ACTION Ca_StandbySub4:
IF Mach_Control.U.DT_iMode=1 THEN//在自动状态下	
//Ca_Step3-----负极叠片搬运取纠偏位极片
CASE Ca_Step3 OF
	10:
		IF arrAxisCtrl[AxiseNo.AxisName.CaDTCarryingUpDown].Status.Enabled AND arrAxisCtrl[AxiseNo.AxisName.CaDTCarryingLine].Status.Enabled  THEN
			arrCyCtrl[arrCyNo.CylinderName.CaScrapbinCy].Cmd.bON:=TRUE;//负极纠偏NG料盒气缸伸出
			IF arrCyCtrl[arrCyNo.CylinderName.CaScrapbinCy].Status.ONState THEN
				arrCyCtrl[arrCyNo.CylinderName.CaScrapbinUDCy].Cmd.bOFF:=TRUE;//负极纠偏NG料盒气缸升降气缸下降
				IF  arrCyCtrl[arrCyNo.CylinderName.CaScrapbinUDCy].Status.OFFState THEN
					Ca_Step3:=11;
				END_IF
			END_IF	
		END_IF
	11://判断负极搬运平移2是否在初始位，负极搬运升降2上升至初始高度、负极叠片升降上升至初始高度
		IF arrAxisCtrl[AxiseNo.AxisName.CaDTCarryingLine].Cmd.arrbRealPoint[1] THEN
			IF Mach_Control.DT_b.SinStepMode THEN//单步调试模式
				DP_SinStepe:=TRUE;
			ELSE
				DP_SinStepe:=FALSE;	
			END_IF			
			Ca_Step3:=30;
		ELSE
			IF arrAxisCtrl[AxiseNo.AxisName.CaDTCarryingUpDown].Status.Homed AND arrAxisCtrl[AxiseNo.AxisName.CaDTCarryingUpDown].Status.NoMoving AND
				NOT arrAxisCtrl[AxiseNo.AxisName.CaDTCarryingUpDown].Status.Error THEN
				IF arrAxisCtrl[AxiseNo.AxisName.CaDTCarryingUpDown].Cmd.arrbRealPoint[4] THEN
					arrAxisCtrl[AxiseNo.AxisName.CaDTCarryingUpDown].Cmd.iGoSetPos:=0;
					IF Mach_Control.DT_b.SinStepMode THEN//单步调试模式
						DP_SinStepe:=TRUE;
					ELSE
						DP_SinStepe:=FALSE;	
					END_IF								
					Ca_Step3:=20;
				ELSE
					arrAxisCtrl[AxiseNo.AxisName.CaDTCarryingUpDown].Cmd.iGoSetPos:=4;//负极叠片升降移动至等待高度
				END_IF
			END_IF
		END_IF
	20://负极叠片搬运平移至初始位，负极搬运在安全位
		//IF arrAxisCtrl[AxiseNo.AxisName.CaDTCarryingLine].Status.fActPos < (arrAxisPar[AxiseNo.AxisName.CaDTCarryingLine].arrTargetPoint[2]-180) THEN
			//arrCyCtrl[arrCyNo.ElectValveName.CadeviationIonizedWind].Cmd.bON:=TRUE;//负极纠偏平台除尘
			//arrCyCtrl[arrCyNo.ElectValveName.CadeviationIonizedWind].Cmd.bOFF:=FALSE;//负极纠偏平台除尘
		//END_IF	
		IF NOT DP_SinStepe THEN
			//arrCyCtrl[arrCyNo.CylinderName.CaScrapbinCy].Cmd.bOFF:=TRUE;//负极纠偏NG料盒气缸收回   Mach_Control.Ca_b.CarryingSafepos[0] 
			IF TailCurlSEPTA_SafePos AND arrAxisCtrl[AxiseNo.AxisName.CaCarryingUpDown2].Cmd.arrbRealPoint[4] AND arrAxisCtrl[AxiseNo.AxisName.CaDTCarryingUpDown].Cmd.arrbRealPoint[4] AND arrAxisCtrl[AxiseNo.AxisName.CaDTCarryingLine].Status.Homed AND
				arrAxisCtrl[AxiseNo.AxisName.CaDTCarryingLine].Status.NoMoving AND NOT arrAxisCtrl[AxiseNo.AxisName.CaDTCarryingLine].Status.Error (*AND NOT arrAxisCtrl[AxiseNo.AxisName.CaCarryingLine2].Status.Error AND
				arrAxisCtrl[AxiseNo.AxisName.CaCarryingLine2].Status.fActPos < arrAxisPar[AxiseNo.AxisName.CaCarryingLine2].arrTargetPoint[2]*)    THEN
				IF arrAxisCtrl[AxiseNo.AxisName.CaDTCarryingLine].Cmd.arrbRealPoint[1] THEN
					Ca_DTCarryingTorMark:=FALSE;//负极叠台搬运平移力矩判断标志位
					arrAxisCtrl[AxiseNo.AxisName.CaDTCarryingLine].Cmd.iGoSetPos:=0;
					IF Mach_Control.DT_b.SinStepMode THEN//单步调试模式
						DP_SinStepe:=TRUE;
					ELSE
						DP_SinStepe:=FALSE;	
					END_IF					
					Ca_Step3:=30;
				ELSE
					arrAxisCtrl[AxiseNo.AxisName.CaDTCarryingLine].Cmd.iGoSetPos:=1;//负极叠片平移至初始位
					Ca_DTCarryingTorMark:=TRUE;//负极叠台搬运平移力矩判断标志位
				END_IF
			END_IF
		END_IF
	30://判断纠偏平台是否允许取极片
		IF NOT DP_SinStepe THEN
			IF 	Mach_Control.Ca_b.Ca_deviationDPOK OR Mach_Control.U.EmptyRunMode  THEN
				IF Mach_Control.DT_b.SinStepMode THEN//单步调试模式
					DP_SinStepe:=TRUE;
				ELSE
					DP_SinStepe:=FALSE;	
				END_IF			
				IF Mach_Control.DT_b.DT_CCD_TwoModel THEN
					CCD.CaRec.Finish.RectifyX1:=0;
					CCD.CaRec.Finish.RectifyX2:=0;
					CCD.CaRec.Finish.RectifyY:=0;		
					CCD.CaRec.Finish.RectifyResult:=0;//拍照结果清零									
					Mach_Control.Ca_b.Ca_CCDStart :=TRUE;//启动CCD拍照
					CCD.CaRec.Start.iPhotoDo:=2;//启动CCD第二次拍照
				END_IF		
				Ca_TON[7].IN:=FALSE;
				Ca_Step3:=40;
			END_IF
		END_IF
	
END_CASE
END_IF



CASE Ca_Step3 OF

	40://AND  arrCyCtrl[arrCyNo.CylinderName.CaScrapbinCy].Io.DIOFFSwitch  arrCyCtrl[arrCyNo.CylinderName.CaScrapbinCy].Io.DIOFFSwitch AND						
		IF NOT DP_SinStepe THEN
			arrCyCtrl[arrCyNo.ElectValveName.CaDTCarryingVacuum].Cmd.bON:=FALSE;//负极叠片搬运升降真空开
			arrCyCtrl[arrCyNo.ElectValveName.CaDTCarryingVacuum].Cmd.bOFF:=TRUE;//负极叠片搬运升降真空开
	
			//arrCyCtrl[arrCyNo.CylinderName.CaScrapbinCy].Cmd.bOFF:=TRUE;//负极纠偏NG料盒气缸收回
			IF  arrAxisCtrl[AxiseNo.AxisName.CaDTCarryingUpDown].Status.Homed AND 
				arrAxisCtrl[AxiseNo.AxisName.CaDTCarryingUpDown].Status.NoMoving AND NOT arrAxisCtrl[AxiseNo.AxisName.CaDTCarryingUpDown].Status.Error THEN
				IF arrAxisCtrl[AxiseNo.AxisName.CaDTCarryingUpDown].Cmd.arrbRealPoint[2] AND arrCyCtrl[arrCyNo.CylinderName.CaScrapbinCy].Status.ONState THEN
					arrCyCtrl[arrCyNo.ElectValveName.CadeviationVacuum].Cmd.bOFF:=TRUE;//负极纠偏平台真空关闭
					arrCyCtrl[arrCyNo.ElectValveName.CadeviationVacuum].Cmd.bON:=FALSE;//负极纠偏平台真空关闭
					arrCyCtrl[arrCyNo.ElectValveName.CadeviationVacuumBark].Cmd.bON:=TRUE;//负极纠偏平台破真空打开	
					arrCyCtrl[arrCyNo.ElectValveName.CadeviationVacuumBark].Cmd.bOFF:=FALSE;//负极纠偏平台破真空打开		
					//IF Mach_Control.Ca_b.Ca_deviationFalg THEN
						Mach_Control.Ca_b.Ca_DPCarryingFalg:=TRUE;//置位叠片真空吸盘有料标记	
						Mach_Control.Ca_b.Ca_deviationFalg:=FALSE;//复位纠偏平台有料标记			
					//END_IF
					Par.stDT_date.Ca_MQ_Slice[9]:=Par.stDT_date.Ca_MQ_Slice[8];											
					arrAxisCtrl[AxiseNo.AxisName.CaDTCarryingUpDown].Cmd.iGoSetPos:=0;									
					IF NOT Ca_TON[7].Q THEN
						Ca_TON[7].IN:=TRUE;
					ELSE
						IF Mach_Control.DT_b.SinStepMode THEN//单步调试模式
							DP_SinStepe:=TRUE;
						ELSE
							DP_SinStepe:=FALSE;	
						END_IF			
						Ca_TON[7].IN:=FALSE;
						Ca_Step3:=50;												
					END_IF												
				ELSE
					arrAxisCtrl[AxiseNo.AxisName.CaDTCarryingUpDown].Cmd.iGoSetPos:=2;//负极叠片升降下降至取纠偏极片高度
				END_IF
			END_IF	
		END_IF
	50://负极叠片搬运升降上升至凸轮耦合初始位
		IF arrAxisCtrl[AxiseNo.AxisName.CaDTCarryingUpDown].Status.Homed AND arrAxisCtrl[AxiseNo.AxisName.CaDTCarryingUpDown].Status.NoMoving AND 
			NOT arrAxisCtrl[AxiseNo.AxisName.CaDTCarryingUpDown].Status.Error THEN
				IF arrAxisCtrl[AxiseNo.AxisName.CaDTCarryingUpDown].Cmd.arrbRealPoint[4] THEN
					arrAxisCtrl[AxiseNo.AxisName.CaDTCarryingUpDown].Cmd.iGoSetPos:=0;
					Ca_Step3:=6666;
				ELSE
					arrAxisCtrl[AxiseNo.AxisName.CaDTCarryingUpDown].Cmd.iGoSetPos:=4;//负极叠片升降移动至初始高度
				END_IF
		END_IF		
END_CASE
END_ACTION

ACTION Code:
(*
 TJ_Scan_M(CLK:=Mach_Control.TJ_b.Scan_CT , Q=> );
 CASE scan_Step OF
	0:
		IF TJ_Scan_M.Q THEN
			scan_Step:=5;
		END_IF
	5:
		 Mach_Control.TJ_b.Scan_Men[4]:=Mach_Control.TJ_b.Scan_Men[3];
		 scan_Step:=10;
	 
	10:
		Mach_Control.TJ_b.Scan_Men[3]:=Mach_Control.TJ_b.Scan_Men[2];
	 	scan_Step:=20;
	 
	 20:
	 	Mach_Control.TJ_b.Scan_Men[2]:=Mach_Control.TJ_b.Scan_Men[1];
	 	scan_Step:=30;
	 
	 30:
	 		Mach_Control.TJ_b.Scan_Men[1].Scan_gross:=Mach_Control.TJ_b.Scan_gross;
	 		Mach_Control.TJ_b.Scan_Men[1].TJ_Code:=Mach_Control.TJ_b.strCode;
	 		scan_Step:=0;
	 
	 
 END_CASE
 *)
END_ACTION

ACTION Dietai_Cam:
DT_Cam_ton[1](PT:=T#100MS);
DT_Cam_ton[2](PT:=T#100MS);
DT_Cam_ton[3](PT:=T#100MS);
DT_Cam_ton[4](PT:=T#100MS);
DT_Cam_ton[5](PT:=T#100MS);
DT_Cam_ton[5](PT:=T#100MS);//
(***********************************压刀凸轮表创建************************************************)
(*
    fbCrectCamLeftYDLine                   :FB_CrectCamYaDaoLine ;
     fbCrectCamLeftYDUpDown             :FB_CrectCamYaDaoUpDown ;
     fbCrectCamRightYDLine                 :FB_CrectCamYaDaoLine ;
     fbCrectCamRightYDUpDown           :FB_CrectCamYaDaoUpDown ;
*)
//左压刀升降凸轮创建 
//fbCrectCamLeftYDUpDown.fMoveLength:=-ABS(arrAxisPar[AxiseNo.AxisName.LeftYDUpDown].arrTargetPoint[1]-arrAxisPar[AxiseNo.AxisName.LeftYDUpDown].arrTargetPoint[2]);
//fbCrectCamLeftYDUpDown.fSaveLength1:=-ABS(arrAxisPar[AxiseNo.AxisName.LeftYDUpDown].arrTargetPoint[1]-arrAxisPar[AxiseNo.AxisName.LeftYDUpDown].arrTargetPoint[3]);
fbCrectCamLeftYDUpDown.fMoveLength:=-ABS(arrAxisPar[AxiseNo.AxisName.LeftYDUpDown].arrTargetPoint[11]+arrAxisPar[AxiseNo.AxisName.LeftYDUpDown].arrTargetPoint[13]);
fbCrectCamLeftYDUpDown.fSaveLength1:=-ABS(arrAxisPar[AxiseNo.AxisName.LeftYDUpDown].arrTargetPoint[12]+arrAxisPar[AxiseNo.AxisName.LeftYDUpDown].arrTargetPoint[13]);
fbCrectCamLeftYDUpDown.fSaveLength2:=-3;

fbCrectCamLeftYDUpDown(
	bCreatTable:=                       fbCrectCamLeftYDUpDown.bCreatTable , 
	Reset:=                                 stSysState.bReset  ,  
	iTable:=                                TableNo.M_LeftYDUpDown  , 
	fMoveLength:=  , //压刀升降最大高度
	fSaveLength1:= , //压刀抽刀高度
	fSaveLength2:= , //压刀下压高度
	fMasterKeyPos1:=240 , //220 240
	fMasterKeyPos2:=258 , //234 250
	fMasterKeyPos3:=275 , //252 255
	fMasterKeyPos4:=307 , //300
	//fMasterKeyPos5:=313 , //330
	fMasterKeyPos6:=342 , //342
    axisMaster:=                          arrAxis[AxiseNo.VirAxisName.VirMain] ,   
	axisSlave:=                             arrAxis[AxiseNo.AxisName.LeftYDUpDown] ,  
	
	bCreatTableDone=> , 
	bCreatTableError=> , 
	bError=> );
fbCrectCamLeftYDUpDown.bCreatTableDone;
fbCrectCamLeftYDUpDown.bCreatTableError;
fbCrectCamLeftYDUpDown.bError;

//左压刀开合凸轮创建
//fbCrectCamLeftYDLine.fMoveLength:=-ABS(arrAxisPar[AxiseNo.AxisName.LeftYDLine].arrTargetPoint[1]-arrAxisPar[AxiseNo.AxisName.LeftYDLine].arrTargetPoint[2]);
fbCrectCamLeftYDLine.fMoveLength:=-ABS(arrAxisPar[AxiseNo.AxisName.LeftYDLine].arrTargetPoint[11]);
fbCrectCamLeftYDLine.fMoveLength2:=-ABS(arrAxisPar[AxiseNo.AxisName.LeftYDLine].arrTargetPoint[12]);	
fbCrectCamLeftYDLine(
	bCreatTable:=                         fbCrectCamLeftYDLine.bCreatTable , 
	Reset:=                                   stSysState.bReset  ,  
	iTable:=                                   TableNo.M_LeftYDLine  , 
	fMoveLength:= , 
	fMasterKeyPos1:=260 , //234  250
	fMasterKeyPos4:=40 , //234  250
	fMasterKeyPos2:=293 , //290
	fMasterKeyPos3:=328 , //324
	axisMaster:=                       arrAxis[AxiseNo.VirAxisName.VirMain] ,   
    axisSlave:=                          arrAxis[AxiseNo.AxisName.LeftYDLine] ,  
	bCreatTableDone=>  , 
	bCreatTableError=> , 
	bError=> );
fbCrectCamLeftYDLine.bCreatTableDone;
fbCrectCamLeftYDLine.bCreatTableError;
fbCrectCamLeftYDLine.bError;

//右压刀开合
//fbCrectCamRightYDLine.fMoveLength:=-ABS(arrAxisPar[AxiseNo.AxisName.RightYDLine].arrTargetPoint[1]-arrAxisPar[AxiseNo.AxisName.RightYDLine].arrTargetPoint[2]);
fbCrectCamRightYDLine.fMoveLength:=-ABS(arrAxisPar[AxiseNo.AxisName.RightYDLine].arrTargetPoint[11]);
fbCrectCamRightYDLine.fMoveLength2:=-ABS(arrAxisPar[AxiseNo.AxisName.RightYDLine].arrTargetPoint[12]);
fbCrectCamRightYDLine(
	bCreatTable:=                         fbCrectCamRightYDLine.bCreatTable , 
	Reset:=                                   stSysState.bReset  ,  
	iTable:=                                   TableNo.M_RightYDLine  , 
	fMoveLength:= , 

	fMasterKeyPos1:=260 , //234  250
	fMasterKeyPos4:=40 , //234  250
	fMasterKeyPos2:=293 ,//290
	fMasterKeyPos3:=328 , //324

	axisMaster:=                       arrAxis[AxiseNo.VirAxisName.VirMain] ,   
    axisSlave:=                          arrAxis[AxiseNo.AxisName.RightYDLine] ,  
	bCreatTableDone=>  , 
	bCreatTableError=> , 
	bError=> );
fbCrectCamRightYDLine.bCreatTableDone;
fbCrectCamRightYDLine.bCreatTableError;
fbCrectCamRightYDLine.bError;

//右压刀升降凸轮创建
//fbCrectCamRightYDUpDown.fMoveLength:=-ABS(arrAxisPar[AxiseNo.AxisName.RightYDUpDown].arrTargetPoint[1]-arrAxisPar[AxiseNo.AxisName.RightYDUpDown].arrTargetPoint[2]);
//fbCrectCamRightYDUpDown.fSaveLength1:=-ABS(arrAxisPar[AxiseNo.AxisName.RightYDUpDown].arrTargetPoint[1]-arrAxisPar[AxiseNo.AxisName.RightYDUpDown].arrTargetPoint[3]);
fbCrectCamRightYDUpDown.fMoveLength:=-ABS(arrAxisPar[AxiseNo.AxisName.RightYDUpDown].arrTargetPoint[11]+arrAxisPar[AxiseNo.AxisName.RightYDUpDown].arrTargetPoint[13]);
fbCrectCamRightYDUpDown.fSaveLength1:=-ABS(arrAxisPar[AxiseNo.AxisName.RightYDUpDown].arrTargetPoint[12]+arrAxisPar[AxiseNo.AxisName.RightYDUpDown].arrTargetPoint[13]);	
fbCrectCamRightYDUpDown.fSaveLength2:=-3;
fbCrectCamRightYDUpDown(
	bCreatTable:=                       fbCrectCamRightYDUpDown.bCreatTable , 
	Reset:=                                 stSysState.bReset  ,  
	iTable:=                                TableNo.M_RightYDUpDown  , 
	fMoveLength:= , 
	fSaveLength1:= , 
	fSaveLength2:= ,
	fMasterKeyPos1:=240 , //220 240
	fMasterKeyPos2:=258 , //234 250
	fMasterKeyPos3:=275 , //252 255
	fMasterKeyPos4:=307 , //300
	//fMasterKeyPos5:=313 , //330
	fMasterKeyPos6:=342 , //342
    axisMaster:=                          arrAxis[AxiseNo.VirAxisName.VirMain] ,   
	axisSlave:=                             arrAxis[AxiseNo.AxisName.RightYDUpDown] ,  
	
	bCreatTableDone=> , 
	bCreatTableError=> , 
	bError=> );
fbCrectCamRightYDUpDown.bCreatTableDone;
fbCrectCamRightYDUpDown.bCreatTableError;
fbCrectCamRightYDUpDown.bError;


//左压刀升降凸轮创建 2
fbCrectCamLeftYDUpDown2.fMoveLength:=-ABS(arrAxisPar[AxiseNo.AxisName.LeftYDUpDown].arrTargetPoint[11]+arrAxisPar[AxiseNo.AxisName.LeftYDUpDown].arrTargetPoint[13]);
fbCrectCamLeftYDUpDown2.fSaveLength1:=-ABS(arrAxisPar[AxiseNo.AxisName.LeftYDUpDown].arrTargetPoint[11]+arrAxisPar[AxiseNo.AxisName.LeftYDUpDown].arrTargetPoint[13]);
fbCrectCamLeftYDUpDown2.fSaveLength2:=ABS(arrAxisPar[AxiseNo.AxisName.LeftYDUpDown].arrTargetPoint[12]+arrAxisPar[AxiseNo.AxisName.LeftYDUpDown].arrTargetPoint[13]);
fbCrectCamLeftYDUpDown2(
	bCreatTable:=                       fbCrectCamLeftYDUpDown2.bCreatTable , 
	Reset:=                                 stSysState.bReset  ,  
	iTable:=                                TableNo.M_LeftYDUpDown2  , 
	fMoveLength:=  , //压刀升降最大高度
	fSaveLength1:= , //压刀抽刀高度
	fSaveLength2:= , //
	fMasterKeyPos1:=260 , //240
	fMasterKeyPos2:=300 , //234 250
	fMasterKeyPos3:=301 , //252 255
	fMasterKeyPos4:=302 , //300
//	fMasterKeyPos5:=342 , //300
    fMasterKeyPos6:=342 , //342
    axisMaster:=                          arrAxis[AxiseNo.VirAxisName.VirMain] ,   
	axisSlave:=                             arrAxis[AxiseNo.AxisName.LeftYDUpDown] ,  
	
	bCreatTableDone=> , 
	bCreatTableError=> , 
	bError=> );
fbCrectCamLeftYDUpDown2.bCreatTableDone;
fbCrectCamLeftYDUpDown2.bCreatTableError;
fbCrectCamLeftYDUpDown.bError;

//左压刀开合凸轮创建2

fbCrectCamLeftYDLine2.fMoveLength:=ABS(arrAxisPar[AxiseNo.AxisName.LeftYDLine].arrTargetPoint[1]-arrAxisPar[AxiseNo.AxisName.LeftYDLine].arrTargetPoint[2]);
fbCrectCamLeftYDLine2(
	bCreatTable:=                         fbCrectCamLeftYDLine2.bCreatTable , 
	Reset:=                                   stSysState.bReset  ,  
	iTable:=                                   TableNo.M_LeftYDLine2  , 
	fMoveLength:= , 
	fMasterKeyPos1:=285 , //234  250
	fMasterKeyPos4:=40 , //234  250
	fMasterKeyPos2:=293 , //290
	fMasterKeyPos3:=328 , //324
	axisMaster:=                       arrAxis[AxiseNo.VirAxisName.VirMain] ,   
    axisSlave:=                          arrAxis[AxiseNo.AxisName.LeftYDLine] ,  
	bCreatTableDone=>  , 
	bCreatTableError=> , 
	bError=> );
fbCrectCamLeftYDLine2.bCreatTableDone;
fbCrectCamLeftYDLine2.bCreatTableError;
fbCrectCamLeftYDLine2.bError;


//右压刀开合2

fbCrectCamRightYDLine2.fMoveLength:=ABS(arrAxisPar[AxiseNo.AxisName.RightYDLine].arrTargetPoint[1]-arrAxisPar[AxiseNo.AxisName.RightYDLine].arrTargetPoint[2]);
fbCrectCamRightYDLine2(
	bCreatTable:=                         fbCrectCamRightYDLine2.bCreatTable , 
	Reset:=                                   stSysState.bReset  ,  
	iTable:=                                   TableNo.M_RightYDLine2  , 
	fMoveLength:= , 

	fMasterKeyPos1:=285 , //234  250
	fMasterKeyPos4:=40 , //234  250
	fMasterKeyPos2:=293 ,//290
	fMasterKeyPos3:=328 , //324

	axisMaster:=                       arrAxis[AxiseNo.VirAxisName.VirMain] ,   
    axisSlave:=                          arrAxis[AxiseNo.AxisName.RightYDLine] ,  
	bCreatTableDone=>  , 
	bCreatTableError=> , 
	bError=> );
fbCrectCamRightYDLine2.bCreatTableDone;
fbCrectCamRightYDLine2.bCreatTableError;
fbCrectCamRightYDLine2.bError;

//右压刀升降凸轮创建2
fbCrectCamRightYDUpDown2.fMoveLength:=-ABS(arrAxisPar[AxiseNo.AxisName.RightYDUpDown].arrTargetPoint[11]+arrAxisPar[AxiseNo.AxisName.RightYDUpDown].arrTargetPoint[13]);
fbCrectCamRightYDUpDown2.fSaveLength1:=-ABS(arrAxisPar[AxiseNo.AxisName.RightYDUpDown].arrTargetPoint[11]+arrAxisPar[AxiseNo.AxisName.RightYDUpDown].arrTargetPoint[13]);	
fbCrectCamRightYDUpDown2.fSaveLength2:=ABS(arrAxisPar[AxiseNo.AxisName.RightYDUpDown].arrTargetPoint[12]+arrAxisPar[AxiseNo.AxisName.RightYDUpDown].arrTargetPoint[13]);
fbCrectCamRightYDUpDown2(
	bCreatTable:=                       fbCrectCamRightYDUpDown2.bCreatTable , 
	Reset:=                                 stSysState.bReset  ,  
	iTable:=                                TableNo.M_RightYDUpDown2  , 
	fMoveLength:= , 
	fSaveLength1:= , 
	fSaveLength2:= ,
	fMasterKeyPos1:=260 , //240
	fMasterKeyPos2:=300 , //234 250
	fMasterKeyPos3:=301 , //252 255
	fMasterKeyPos4:=302 , //300
//	fMasterKeyPos5:=342 , //300
    fMasterKeyPos6:=342 , //342
    axisMaster:=                          arrAxis[AxiseNo.VirAxisName.VirMain] ,   
	axisSlave:=                             arrAxis[AxiseNo.AxisName.RightYDUpDown] ,  
	
	bCreatTableDone=> , 
	bCreatTableError=> , 
	bError=> );
fbCrectCamRightYDUpDown2.bCreatTableDone;
fbCrectCamRightYDUpDown2.bCreatTableError;
fbCrectCamRightYDUpDown2.bError;

tYDCreateCamTON(IN:= , PT:=T#0.5S , Q=> , ET=> );
IF Mach_Control.U.DT_iMode=3 OR Mach_Control.U.DT_iMode=0 THEN//在手动状态下
			//从触摸屏创建叠台压刀凸轮
			rYDCreateCam_TRIG(CLK:=Mach_Control.DT_b.CreateCamStart1 , Q=> );		
			IF rYDCreateCam_TRIG.Q THEN
				tYDCreateCamTON.IN:=FALSE;
				YDCrectCamStep0:=10;
				Mach_Control.DT_b.Error[0]:=FALSE;
			END_IF
END_IF			
			//叠台压刀凸轮自动创建
			CASE YDCrectCamStep0 OF
					10:
							IF NOT 	tYDCreateCamTON.Q THEN
									fbCrectCamLeftYDUpDown.bCreatTable:=FALSE;;//左压刀升降凸轮创建
									fbCrectCamLeftYDLine.bCreatTable:=FALSE;//左压刀开合凸轮创建
									fbCrectCamRightYDLine.bCreatTable :=FALSE;//右压刀开合凸轮创建
									 fbCrectCamRightYDUpDown.bCreatTable:=FALSE;//右压刀升降凸轮创建
									 Mach_Control.DT_b.CreateCamDone1:=FALSE;	
									 tYDCreateCamTON.IN:=TRUE;				
							ELSE
										tYDCreateCamTON.IN:=FALSE;
										YDCrectCamStep0:=11;
							END_IF
							
					11:
							IF  NOT DT_Cam_ton[1].Q THEN
								arrAxisCtrl[AxiseNo.AxisName.LeftYDLine].Cmd.bStop:=TRUE;
								arrAxisCtrl[AxiseNo.AxisName.LeftYDUpDown].Cmd.bStop:=TRUE;
								arrAxisCtrl[AxiseNo.AxisName.RightYDLine].Cmd.bStop:=TRUE;
								arrAxisCtrl[AxiseNo.AxisName.RightYDUpDown].Cmd.bStop:=TRUE;
								DT_Cam_ton[1].IN:=TRUE;
							ELSE
								DT_Cam_ton[1].IN:=FALSE;
								YDCrectCamStep0:=12;
								arrAxisCtrl[AxiseNo.AxisName.LeftYDLine].Cmd.bStop:=FALSE;
								arrAxisCtrl[AxiseNo.AxisName.LeftYDUpDown].Cmd.bStop:=FALSE;
								arrAxisCtrl[AxiseNo.AxisName.RightYDLine].Cmd.bStop:=FALSE;
								arrAxisCtrl[AxiseNo.AxisName.RightYDUpDown].Cmd.bStop:=FALSE;
							END_IF
					
					12:
						IF  NOT DT_Cam_ton[2].Q THEN
							arrAxisCtrl[AxiseNo.AxisName.LeftYDLine].Cmd.bReset:=TRUE;	
							arrAxisCtrl[AxiseNo.AxisName.LeftYDUpDown].Cmd.bReset:=TRUE;
							arrAxisCtrl[AxiseNo.AxisName.RightYDLine].Cmd.bReset:=TRUE;
							arrAxisCtrl[AxiseNo.AxisName.RightYDUpDown].Cmd.bReset:=TRUE;		
							DT_Cam_ton[2].IN:=TRUE;
						 ELSE
							 DT_Cam_ton[2].IN:=FALSE;
							 YDCrectCamStep0:=13;
							arrAxisCtrl[AxiseNo.AxisName.LeftYDLine].Cmd.bReset:=FALSE;	
							arrAxisCtrl[AxiseNo.AxisName.LeftYDUpDown].Cmd.bReset:=FALSE;
							arrAxisCtrl[AxiseNo.AxisName.RightYDLine].Cmd.bReset:=FALSE;
							arrAxisCtrl[AxiseNo.AxisName.RightYDUpDown].Cmd.bReset:=FALSE;	
						 END_IF
							
					13:
						arrAxisCtrl[AxiseNo.AxisName.LeftYDLine].Cmd.bEnable:=TRUE;
						arrAxisCtrl[AxiseNo.AxisName.LeftYDUpDown].Cmd.bEnable:=TRUE;
						arrAxisCtrl[AxiseNo.AxisName.RightYDLine].Cmd.bEnable:=TRUE;
						arrAxisCtrl[AxiseNo.AxisName.RightYDUpDown].Cmd.bEnable:=TRUE;
						
						IF arrAxisCtrl[AxiseNo.AxisName.LeftYDLine].Status.Enabled AND arrAxisCtrl[AxiseNo.AxisName.LeftYDUpDown].Status.Enabled AND
							arrAxisCtrl[AxiseNo.AxisName.RightYDLine].Status.Enabled AND arrAxisCtrl[AxiseNo.AxisName.RightYDUpDown].Status.Enabled THEN
							 YDCrectCamStep0:=20;
						END_IF		
				
							
					20://创建凸轮
						fbCrectCamLeftYDUpDown.bCreatTable:=TRUE;;//左压刀升降凸轮创建
						fbCrectCamLeftYDLine.bCreatTable:=TRUE;//左压刀开合凸轮创建
						fbCrectCamRightYDLine.bCreatTable :=TRUE;//右压刀开合凸轮创建
						 fbCrectCamRightYDUpDown.bCreatTable:=TRUE;//右压刀升降凸轮创建
						fbCrectCamLeftYDUpDown2.bCreatTable:=TRUE;;//左压刀升降凸轮创建2
						fbCrectCamLeftYDLine2.bCreatTable:=TRUE;//左压刀开合凸轮创建2
						fbCrectCamRightYDLine2.bCreatTable :=TRUE;//右压刀开合凸轮创建2
						 fbCrectCamRightYDUpDown2.bCreatTable:=TRUE;//右压刀升降凸轮创建	2							 
						 Mach_Control.DT_b.CreateCamDone1:=FALSE;
						 YDCrectCamStep0:=30;
					30://等待凸轮创建完成
						IF fbCrectCamLeftYDUpDown.bCreatTableDone AND fbCrectCamLeftYDLine.bCreatTableDone AND fbCrectCamRightYDLine.bCreatTableDone AND fbCrectCamRightYDUpDown.bCreatTableDone AND
                          fbCrectCamLeftYDUpDown2.bCreatTableDone AND fbCrectCamLeftYDLine2.bCreatTableDone AND fbCrectCamRightYDLine2.bCreatTableDone AND fbCrectCamRightYDUpDown2.bCreatTableDone  THEN
								Mach_Control.DT_b.CreateCamDone1:=TRUE;//叠台压凸轮创建完成
								YDCrectCamStep0:=6666;
						ELSE
								IF fbCrectCamLeftYDUpDown.bCreatTableError OR fbCrectCamLeftYDLine.bCreatTableError OR fbCrectCamRightYDLine.bCreatTableError OR fbCrectCamRightYDUpDown.bCreatTableError  OR
                                   fbCrectCamLeftYDUpDown2.bCreatTableError OR fbCrectCamLeftYDLine2.bCreatTableError OR fbCrectCamRightYDLine2.bCreatTableError OR fbCrectCamRightYDUpDown2.bCreatTableError  THEN
									Mach_Control.DT_b.Error[0]:=TRUE;//叠台压刀凸轮创建失败报警
									YDCrectCamStep0:=9999;
								END_IF
						END_IF
			END_CASE


(***********************************压刀凸轮耦合***********************************************)
(*
      fbCamInLeftYDLine                       :FB_CamIn ;    
      fbCamInLeftYDUpDown                :FB_CamIn ;    
      fbCamInRightYDLine                    :FB_CamIn ;    
      fbCamInRightYDUpDown             :FB_CamIn ;    

*)
//左压刀开合凸轮耦合
fbCamInLeftYDLine.ParCamIn.SlaveScaling;
fbCamInLeftYDLine(
	Reset:=                      stSysState.bReset  , 
	bCamInExecute:=       fbCamInLeftYDLine.bCamInExecute, 
	iTable1:=                   TableNo.M_LeftYDLine  , 
	iTable2:=                   TableNo.M_LeftYDLine2, 
	iTableSel:=                 , 
	ParCamIn:= , 
  	axisMaster:=            arrAxis[AxiseNo.VirAxisName.VirMain] ,  
	axisSlave:=               arrAxis[AxiseNo.AxisName.LeftYDLine] ,  
	bError=> , 
	bReady=> , 
	bInSync=> );

Mach_Control.DT_b.Error[12]:=fbCamInLeftYDLine.bError;
fbCamInLeftYDLine.bReady;
fbCamInLeftYDLine.bInSync;

//左压刀升降凸轮耦合
fbCamInLeftYDUpDown.ParCamIn.SlaveScaling;
fbCamInLeftYDUpDown(
	Reset:=                      stSysState.bReset  , 
	bCamInExecute:=       fbCamInLeftYDUpDown.bCamInExecute, 
	iTable1:=                   TableNo.M_LeftYDUpDown  , 
	iTable2:=                   TableNo.M_LeftYDUpDown2 , 
	iTableSel:=                 , 
	ParCamIn:= , 
  	axisMaster:=            arrAxis[AxiseNo.VirAxisName.VirMain] ,  
	axisSlave:=               arrAxis[AxiseNo.AxisName.LeftYDUpDown] ,  
	bError=> , 
	bReady=> , 
	bInSync=> );

Mach_Control.DT_b.Error[13]:=fbCamInLeftYDUpDown.bError;
fbCamInLeftYDUpDown.bReady;
fbCamInLeftYDUpDown.bInSync;



//右压刀开合凸轮耦合
fbCamInRightYDLine.ParCamIn.SlaveScaling;
fbCamInRightYDLine(
	Reset:=                      stSysState.bReset  , 
	bCamInExecute:=       fbCamInRightYDLine.bCamInExecute, 
	iTable1:=                   TableNo.M_RightYDLine  , 
	iTable2:=                   TableNo.M_RightYDLine2, 
	iTableSel:=                 , 
	ParCamIn:= , 
  	axisMaster:=            arrAxis[AxiseNo.VirAxisName.VirMain] ,  
	axisSlave:=               arrAxis[AxiseNo.AxisName.RightYDLine] ,  
	bError=> , 
	bReady=> , 
	bInSync=> );

Mach_Control.DT_b.Error[14]:=fbCamInRightYDLine.bError;
fbCamInRightYDLine.bReady;
fbCamInRightYDLine.bInSync;


//右压刀升降凸轮耦合
fbCamInRightYDUpDown.ParCamIn.SlaveScaling;
fbCamInRightYDUpDown(
	Reset:=                      stSysState.bReset  , 
	bCamInExecute:=       fbCamInRightYDUpDown.bCamInExecute, 
	iTable1:=                   TableNo.M_RightYDUpDown  , 
	iTable2:=                   TableNo.M_RightYDUpDown2, 
	iTableSel:=                 , 
	ParCamIn:=                , 
  	axisMaster:=            arrAxis[AxiseNo.VirAxisName.VirMain] ,  
	axisSlave:=               arrAxis[AxiseNo.AxisName.RightYDUpDown] ,  
	bError=> , 
	bReady=> , 
	bInSync=> );

Mach_Control.DT_b.Error[15]:=fbCamInRightYDUpDown.bError;
fbCamInRightYDUpDown.bReady;
fbCamInRightYDUpDown.bInSync;
















(*

(*********************************BAK   V1 20240312************************************************)
DT_Cam_ton[1](PT:=T#100MS);
DT_Cam_ton[2](PT:=T#100MS);
DT_Cam_ton[3](PT:=T#100MS);
DT_Cam_ton[4](PT:=T#100MS);
DT_Cam_ton[5](PT:=T#100MS);
DT_Cam_ton[5](PT:=T#100MS);//
(***********************************压刀凸轮表创建************************************************)
(*
    fbCrectCamLeftYDLine                   :FB_CrectCamYaDaoLine ;
     fbCrectCamLeftYDUpDown             :FB_CrectCamYaDaoUpDown ;
     fbCrectCamRightYDLine                 :FB_CrectCamYaDaoLine ;
     fbCrectCamRightYDUpDown           :FB_CrectCamYaDaoUpDown ;
*)
//左压刀升降凸轮创建 
//fbCrectCamLeftYDUpDown.fMoveLength:=-ABS(arrAxisPar[AxiseNo.AxisName.LeftYDUpDown].arrTargetPoint[1]-arrAxisPar[AxiseNo.AxisName.LeftYDUpDown].arrTargetPoint[2]);
//fbCrectCamLeftYDUpDown.fSaveLength1:=-ABS(arrAxisPar[AxiseNo.AxisName.LeftYDUpDown].arrTargetPoint[1]-arrAxisPar[AxiseNo.AxisName.LeftYDUpDown].arrTargetPoint[3]);
fbCrectCamLeftYDUpDown.fMoveLength:=-ABS(arrAxisPar[AxiseNo.AxisName.LeftYDUpDown].arrTargetPoint[11]+arrAxisPar[AxiseNo.AxisName.LeftYDUpDown].arrTargetPoint[13]);
fbCrectCamLeftYDUpDown.fSaveLength1:=-ABS(arrAxisPar[AxiseNo.AxisName.LeftYDUpDown].arrTargetPoint[12]+arrAxisPar[AxiseNo.AxisName.LeftYDUpDown].arrTargetPoint[13]);
fbCrectCamLeftYDUpDown.fSaveLength2:=-3;

fbCrectCamLeftYDUpDown(
	bCreatTable:=                       fbCrectCamLeftYDUpDown.bCreatTable , 
	Reset:=                                 stSysState.bReset  ,  
	iTable:=                                TableNo.M_LeftYDUpDown  , 
	fMoveLength:=  , //压刀升降最大高度
	fSaveLength1:= , //压刀抽刀高度
	fSaveLength2:= , //压刀下压高度
	fMasterKeyPos1:=240 , //220  240
	fMasterKeyPos2:=250 , //234  250
	fMasterKeyPos3:=270 , //252.6  255
	fMasterKeyPos4:=315 , //300.8
	fMasterKeyPos5:=330 , //330
	fMasterKeyPos6:=342 , //342
    axisMaster:=                          arrAxis[AxiseNo.VirAxisName.VirMain] ,   
	axisSlave:=                             arrAxis[AxiseNo.AxisName.LeftYDUpDown] ,  
	
	bCreatTableDone=> , 
	bCreatTableError=> , 
	bError=> );
fbCrectCamLeftYDUpDown.bCreatTableDone;
fbCrectCamLeftYDUpDown.bCreatTableError;
fbCrectCamLeftYDUpDown.bError;

//左压刀开合凸轮创建
//fbCrectCamLeftYDLine.fMoveLength:=-ABS(arrAxisPar[AxiseNo.AxisName.LeftYDLine].arrTargetPoint[1]-arrAxisPar[AxiseNo.AxisName.LeftYDLine].arrTargetPoint[2]);
fbCrectCamLeftYDLine.fMoveLength:=-ABS(arrAxisPar[AxiseNo.AxisName.LeftYDLine].arrTargetPoint[11]);
fbCrectCamLeftYDLine.fMoveLength2:=-ABS(arrAxisPar[AxiseNo.AxisName.LeftYDLine].arrTargetPoint[12]);	
fbCrectCamLeftYDLine(
	bCreatTable:=                         fbCrectCamLeftYDLine.bCreatTable , 
	Reset:=                                   stSysState.bReset  ,  
	iTable:=                                   TableNo.M_LeftYDLine  , 
	fMoveLength:= , 
	fMasterKeyPos1:=250 , //234  250
	fMasterKeyPos4:=270 , //234  250
	fMasterKeyPos2:=290 , //290
	fMasterKeyPos3:=324 , //324
	axisMaster:=                       arrAxis[AxiseNo.VirAxisName.VirMain] ,   
    axisSlave:=                          arrAxis[AxiseNo.AxisName.LeftYDLine] ,  
	bCreatTableDone=>  , 
	bCreatTableError=> , 
	bError=> );
fbCrectCamLeftYDLine.bCreatTableDone;
fbCrectCamLeftYDLine.bCreatTableError;
fbCrectCamLeftYDLine.bError;

//右压刀开合
//fbCrectCamRightYDLine.fMoveLength:=-ABS(arrAxisPar[AxiseNo.AxisName.RightYDLine].arrTargetPoint[1]-arrAxisPar[AxiseNo.AxisName.RightYDLine].arrTargetPoint[2]);
fbCrectCamRightYDLine.fMoveLength:=-ABS(arrAxisPar[AxiseNo.AxisName.RightYDLine].arrTargetPoint[11]);
fbCrectCamRightYDLine.fMoveLength2:=-ABS(arrAxisPar[AxiseNo.AxisName.RightYDLine].arrTargetPoint[12]);
fbCrectCamRightYDLine(
	bCreatTable:=                         fbCrectCamRightYDLine.bCreatTable , 
	Reset:=                                   stSysState.bReset  ,  
	iTable:=                                   TableNo.M_RightYDLine  , 
	fMoveLength:= , 

	fMasterKeyPos1:=250 , //234  250
	fMasterKeyPos4:=270 , //234  250
	fMasterKeyPos2:=290 ,//290
	fMasterKeyPos3:=324 , //324

	axisMaster:=                       arrAxis[AxiseNo.VirAxisName.VirMain] ,   
    axisSlave:=                          arrAxis[AxiseNo.AxisName.RightYDLine] ,  
	bCreatTableDone=>  , 
	bCreatTableError=> , 
	bError=> );
fbCrectCamRightYDLine.bCreatTableDone;
fbCrectCamRightYDLine.bCreatTableError;
fbCrectCamRightYDLine.bError;

//右压刀升降凸轮创建
//fbCrectCamRightYDUpDown.fMoveLength:=-ABS(arrAxisPar[AxiseNo.AxisName.RightYDUpDown].arrTargetPoint[1]-arrAxisPar[AxiseNo.AxisName.RightYDUpDown].arrTargetPoint[2]);
//fbCrectCamRightYDUpDown.fSaveLength1:=-ABS(arrAxisPar[AxiseNo.AxisName.RightYDUpDown].arrTargetPoint[1]-arrAxisPar[AxiseNo.AxisName.RightYDUpDown].arrTargetPoint[3]);
fbCrectCamRightYDUpDown.fMoveLength:=-ABS(arrAxisPar[AxiseNo.AxisName.RightYDUpDown].arrTargetPoint[11]+arrAxisPar[AxiseNo.AxisName.RightYDUpDown].arrTargetPoint[13]);
fbCrectCamRightYDUpDown.fSaveLength1:=-ABS(arrAxisPar[AxiseNo.AxisName.RightYDUpDown].arrTargetPoint[12]+arrAxisPar[AxiseNo.AxisName.RightYDUpDown].arrTargetPoint[13]);	
fbCrectCamRightYDUpDown.fSaveLength2:=-3;
fbCrectCamRightYDUpDown(
	bCreatTable:=                       fbCrectCamRightYDUpDown.bCreatTable , 
	Reset:=                                 stSysState.bReset  ,  
	iTable:=                                TableNo.M_RightYDUpDown  , 
	fMoveLength:= , 
	fSaveLength1:= , 
	fSaveLength2:= ,
	fMasterKeyPos1:=240 , //220 240
	fMasterKeyPos2:=250 , //234 250
	fMasterKeyPos3:=270 , //252 255
	fMasterKeyPos4:=315 , //300
	fMasterKeyPos5:=330 , //330
	fMasterKeyPos6:=342 , //342
    axisMaster:=                          arrAxis[AxiseNo.VirAxisName.VirMain] ,   
	axisSlave:=                             arrAxis[AxiseNo.AxisName.RightYDUpDown] ,  
	
	bCreatTableDone=> , 
	bCreatTableError=> , 
	bError=> );
fbCrectCamRightYDUpDown.bCreatTableDone;
fbCrectCamRightYDUpDown.bCreatTableError;
fbCrectCamRightYDUpDown.bError;

tYDCreateCamTON(IN:= , PT:=T#0.5S , Q=> , ET=> );
IF Mach_Control.U.DT_iMode=3 OR Mach_Control.U.DT_iMode=0 THEN//在手动状态下
			//从触摸屏创建叠台压刀凸轮
			rYDCreateCam_TRIG(CLK:=Mach_Control.DT_b.CreateCamStart1 , Q=> );		
			IF rYDCreateCam_TRIG.Q THEN
				tYDCreateCamTON.IN:=FALSE;
				YDCrectCamStep0:=10;
				Mach_Control.DT_b.Error[0]:=FALSE;
			END_IF
END_IF			
			//叠台压刀凸轮自动创建
			CASE YDCrectCamStep0 OF
					10:
							IF NOT 	tYDCreateCamTON.Q THEN
									fbCrectCamLeftYDUpDown.bCreatTable:=FALSE;;//左压刀升降凸轮创建
									fbCrectCamLeftYDLine.bCreatTable:=FALSE;//左压刀开合凸轮创建
									fbCrectCamRightYDLine.bCreatTable :=FALSE;//右压刀开合凸轮创建
									 fbCrectCamRightYDUpDown.bCreatTable:=FALSE;//右压刀升降凸轮创建
									 Mach_Control.DT_b.CreateCamDone1:=FALSE;	
									 tYDCreateCamTON.IN:=TRUE;				
							ELSE
										tYDCreateCamTON.IN:=FALSE;
										YDCrectCamStep0:=11;
							END_IF
							
					11:
							IF  NOT DT_Cam_ton[1].Q THEN
								arrAxisCtrl[AxiseNo.AxisName.LeftYDLine].Cmd.bStop:=TRUE;
								arrAxisCtrl[AxiseNo.AxisName.LeftYDUpDown].Cmd.bStop:=TRUE;
								arrAxisCtrl[AxiseNo.AxisName.RightYDLine].Cmd.bStop:=TRUE;
								arrAxisCtrl[AxiseNo.AxisName.RightYDUpDown].Cmd.bStop:=TRUE;
								DT_Cam_ton[1].IN:=TRUE;
							ELSE
								DT_Cam_ton[1].IN:=FALSE;
								YDCrectCamStep0:=12;
								arrAxisCtrl[AxiseNo.AxisName.LeftYDLine].Cmd.bStop:=FALSE;
								arrAxisCtrl[AxiseNo.AxisName.LeftYDUpDown].Cmd.bStop:=FALSE;
								arrAxisCtrl[AxiseNo.AxisName.RightYDLine].Cmd.bStop:=FALSE;
								arrAxisCtrl[AxiseNo.AxisName.RightYDUpDown].Cmd.bStop:=FALSE;
							END_IF
					
					12:
						IF  NOT DT_Cam_ton[2].Q THEN
							arrAxisCtrl[AxiseNo.AxisName.LeftYDLine].Cmd.bReset:=TRUE;	
							arrAxisCtrl[AxiseNo.AxisName.LeftYDUpDown].Cmd.bReset:=TRUE;
							arrAxisCtrl[AxiseNo.AxisName.RightYDLine].Cmd.bReset:=TRUE;
							arrAxisCtrl[AxiseNo.AxisName.RightYDUpDown].Cmd.bReset:=TRUE;		
							DT_Cam_ton[2].IN:=TRUE;
						 ELSE
							 DT_Cam_ton[2].IN:=FALSE;
							 YDCrectCamStep0:=13;
							arrAxisCtrl[AxiseNo.AxisName.LeftYDLine].Cmd.bReset:=FALSE;	
							arrAxisCtrl[AxiseNo.AxisName.LeftYDUpDown].Cmd.bReset:=FALSE;
							arrAxisCtrl[AxiseNo.AxisName.RightYDLine].Cmd.bReset:=FALSE;
							arrAxisCtrl[AxiseNo.AxisName.RightYDUpDown].Cmd.bReset:=FALSE;	
						 END_IF
							
					13:
						arrAxisCtrl[AxiseNo.AxisName.LeftYDLine].Cmd.bEnable:=TRUE;
						arrAxisCtrl[AxiseNo.AxisName.LeftYDUpDown].Cmd.bEnable:=TRUE;
						arrAxisCtrl[AxiseNo.AxisName.RightYDLine].Cmd.bEnable:=TRUE;
						arrAxisCtrl[AxiseNo.AxisName.RightYDUpDown].Cmd.bEnable:=TRUE;
						
						IF arrAxisCtrl[AxiseNo.AxisName.LeftYDLine].Status.Enabled AND arrAxisCtrl[AxiseNo.AxisName.LeftYDUpDown].Status.Enabled AND
							arrAxisCtrl[AxiseNo.AxisName.RightYDLine].Status.Enabled AND arrAxisCtrl[AxiseNo.AxisName.RightYDUpDown].Status.Enabled THEN
							 YDCrectCamStep0:=20;
						END_IF		
				
							
					20://创建凸轮
						fbCrectCamLeftYDUpDown.bCreatTable:=TRUE;;//左压刀升降凸轮创建
						fbCrectCamLeftYDLine.bCreatTable:=TRUE;//左压刀开合凸轮创建
						fbCrectCamRightYDLine.bCreatTable :=TRUE;//右压刀开合凸轮创建
						 fbCrectCamRightYDUpDown.bCreatTable:=TRUE;//右压刀升降凸轮创建
						 Mach_Control.DT_b.CreateCamDone1:=FALSE;
						 YDCrectCamStep0:=30;
					30://等待凸轮创建完成
						IF fbCrectCamLeftYDUpDown.bCreatTableDone AND fbCrectCamLeftYDLine.bCreatTableDone AND fbCrectCamRightYDLine.bCreatTableDone AND fbCrectCamRightYDUpDown.bCreatTableDone THEN
								Mach_Control.DT_b.CreateCamDone1:=TRUE;//叠台压凸轮创建完成
								YDCrectCamStep0:=6666;
						ELSE
								IF fbCrectCamLeftYDUpDown.bCreatTableError OR fbCrectCamLeftYDLine.bCreatTableError OR fbCrectCamRightYDLine.bCreatTableError OR fbCrectCamRightYDUpDown.bCreatTableError THEN
									Mach_Control.DT_b.Error[0]:=TRUE;//叠台压刀凸轮创建失败报警
									YDCrectCamStep0:=9999;
								END_IF
						END_IF
			END_CASE


(***********************************压刀凸轮耦合***********************************************)
(*
      fbCamInLeftYDLine                       :FB_CamIn ;    
      fbCamInLeftYDUpDown                :FB_CamIn ;    
      fbCamInRightYDLine                    :FB_CamIn ;    
      fbCamInRightYDUpDown             :FB_CamIn ;    

*)
//左压刀开合凸轮耦合
fbCamInLeftYDLine.ParCamIn.SlaveScaling;
fbCamInLeftYDLine(
	Reset:=                      stSysState.bReset  , 
	bCamInExecute:=       fbCamInLeftYDLine.bCamInExecute, 
	iTable1:=                   TableNo.M_LeftYDLine  , 
	iTable2:=                   , 
	iTableSel:=                 , 
	ParCamIn:= , 
  	axisMaster:=            arrAxis[AxiseNo.VirAxisName.VirMain] ,  
	axisSlave:=               arrAxis[AxiseNo.AxisName.LeftYDLine] ,  
	bError=> , 
	bReady=> , 
	bInSync=> );

Mach_Control.DT_b.Error[12]:=fbCamInLeftYDLine.bError;
fbCamInLeftYDLine.bReady;
fbCamInLeftYDLine.bInSync;

//左压刀升降凸轮耦合
fbCamInLeftYDUpDown.ParCamIn.SlaveScaling;
fbCamInLeftYDUpDown(
	Reset:=                      stSysState.bReset  , 
	bCamInExecute:=       fbCamInLeftYDUpDown.bCamInExecute, 
	iTable1:=                   TableNo.M_LeftYDUpDown  , 
	iTable2:=                   , 
	iTableSel:=                 , 
	ParCamIn:= , 
  	axisMaster:=            arrAxis[AxiseNo.VirAxisName.VirMain] ,  
	axisSlave:=               arrAxis[AxiseNo.AxisName.LeftYDUpDown] ,  
	bError=> , 
	bReady=> , 
	bInSync=> );

Mach_Control.DT_b.Error[13]:=fbCamInLeftYDUpDown.bError;
fbCamInLeftYDUpDown.bReady;
fbCamInLeftYDUpDown.bInSync;



//右压刀开合凸轮耦合
fbCamInRightYDLine.ParCamIn.SlaveScaling;
fbCamInRightYDLine(
	Reset:=                      stSysState.bReset  , 
	bCamInExecute:=       fbCamInRightYDLine.bCamInExecute, 
	iTable1:=                   TableNo.M_RightYDLine  , 
	iTable2:=                   , 
	iTableSel:=                 , 
	ParCamIn:= , 
  	axisMaster:=            arrAxis[AxiseNo.VirAxisName.VirMain] ,  
	axisSlave:=               arrAxis[AxiseNo.AxisName.RightYDLine] ,  
	bError=> , 
	bReady=> , 
	bInSync=> );

Mach_Control.DT_b.Error[14]:=fbCamInRightYDLine.bError;
fbCamInRightYDLine.bReady;
fbCamInRightYDLine.bInSync;


//右压刀升降凸轮耦合
fbCamInRightYDUpDown.ParCamIn.SlaveScaling;
fbCamInRightYDUpDown(
	Reset:=                      stSysState.bReset  , 
	bCamInExecute:=       fbCamInRightYDUpDown.bCamInExecute, 
	iTable1:=                   TableNo.M_RightYDUpDown  , 
	iTable2:=                   , 
	iTableSel:=                 , 
	ParCamIn:=                , 
  	axisMaster:=            arrAxis[AxiseNo.VirAxisName.VirMain] ,  
	axisSlave:=               arrAxis[AxiseNo.AxisName.RightYDUpDown] ,  
	bError=> , 
	bReady=> , 
	bInSync=> );

Mach_Control.DT_b.Error[15]:=fbCamInRightYDUpDown.bError;
fbCamInRightYDUpDown.bReady;
fbCamInRightYDUpDown.bInSync;

*)
END_ACTION

ACTION Dietai_Gohome:
DT_Home_TON[1](PT:=T#0.5S);
DT_Home_TON[2](PT:=T#0.5S);
DT_Home_TON[3](PT:=T#0.5S);


Dietai_GohomeOverTon(IN:= , PT:=T#90S , Q=> , ET=> );//叠台回原点超时报警延时

r_DTinitiStart(CLK:= Mach_Control.DT_b.ALLIniti_Hbtn AND  (TailCurlStep3<>105) AND TailCurlSEPTA_SafePos , Q=> );//叠台部分初始化上升沿
f_DTinitiStart(CLK:= Mach_Control.DT_b.ALLIniti_Hbtn AND  (TailCurlStep3<>105) AND TailCurlSEPTA_SafePos  , Q=> );//叠台部分初始化下降沿

rDT_GohmeTRGI(CLK:=Mach_Control.DT_b.DTIniti_Hbtn , Q=> );//叠台部分初始化上升沿
fDT_GohmeTRGI(CLK:=Mach_Control.DT_b.DTIniti_Hbtn , Q=> );//叠台部分初始化下降沿	
tDT_GohomeTON(IN:= , PT:=T#0.3S , Q=> , ET=> );
Mach_Control.DT_b.ALLIniti_Done:=Mach_Control.Ca_b.Ca_GohomeDone 
AND Mach_Control.An_b.An_GohomeDone  
AND Mach_Control.DT_b.DTIniti_Done 
AND Mach_Control.Ca_b.Ca_BeltGohomeDone ;
////叠片凸轮报警，请初始化叠台后再启动
IF Mach_Control.U.DT_iMode=3 THEN//在手动状态下
		IF r_DTinitiStart.Q THEN
			Mach_Control.DT_b.Step[0]:=0;
			Mach_Control.Ca_b.Ca_GohomeDone:=FALSE;
			Mach_Control.An_b.An_GohomeDone :=FALSE;
			Mach_Control.DT_b.DTIniti_Done:=FALSE;
			Dietai_GohomeDone:=FALSE;//叠台回原点完成
			Dietai_Gohoming:=FALSE;//叠台回原点中
            		Mach_Control.DT_b.DT_camError:=FALSE;//叠片凸轮报警，请初始化叠台后再启动
			//Mach_Control.DT_b.Step[0]:=10;
		END_IF	
END_IF		


IF rDT_GohmeTRGI.Q THEN
	Step_InitDT:=0;
	Dietai_GohomeDone:=FALSE;//叠台回原点完成
	Dietai_Gohoming:=FALSE;//叠台回原点中
	DTIniti_Done:=FALSE;//叠台回原点完成
END_IF	


IF Mach_Control.Ca_b.Ca_GohomeDone AND Mach_Control.An_b.An_GohomeDone AND Mach_Control.DT_b.DTIniti_Done (*AND Mach_Control.Ca_b.Ca_BeltGohomeDone*) THEN
	Mach_Control.DT_b.DT_init_OK:=TRUE;
ELSE
	Mach_Control.DT_b.DT_init_OK:=FALSE;
END_IF
				

(*********************************************************************************叠片轴回原点********************************************************************************************)
IF Mach_Control.U.DT_iMode=3 THEN//在手动状态下
	//回原点超时报警	
	IF  Dietai_Gohoming THEN
		IF  NOT Dietai_GohomeOverTon.Q THEN
			    Dietai_GohomeOverTon.IN:=TRUE;
		ELSE
			IF Dietai_GohomeOverTon.Q THEN
				   Mach_Control. DT_b.Error[23]:=TRUE;//叠台回原点超时报警
				   Dietai_GohomeOverTon.IN:=FALSE;
			END_IF	 			 
		END_IF
	
	ELSE
		Dietai_GohomeOverTon.IN:=FALSE;
	END_IF			

CASE Mach_Control.DT_b.Step[0] OF 
0://在手动模式下触发回原点
	IF f_DTinitiStart.Q THEN
		KD_Mark:=FALSE;//空叠隔膜中	
		DP_CheseCam:=FALSE;
		Step_InitDT:=0;
		Step_InitAnDT:=0;
		Step_InitCaDT:=0;
		Mach_Control.Ca_b.Ca_GohomeDone:=FALSE;
		Mach_Control.An_b.An_GohomeDone :=FALSE;
		Dietai_GohomeDone:=FALSE;//叠台回原点完成
		Mach_Control.An_b.An_GohomeHMI:=FALSE;
		Mach_Control.Ca_b.Ca_GohomeHMI:=FALSE;
		Mach_Control.DT_b.DTIniti_Hbtn:=FALSE;
		Mach_Control.DT_b.DTIniti_Done:=FALSE;
		Blueflaging:=FALSE;	
		Mach_Control.DT_b.Step[0]:=10;
	END_IF
10://正、负极取料初始化
		Mach_Control.An_b.An_GohomeHMI:=TRUE;
		Mach_Control.Ca_b.Ca_GohomeHMI:=TRUE;
		//Mach_Control.DT_b.DT_QLqr:=TRUE;
		Mach_Control.DT_b.Step[0]:=20;	
20://判断正负极取料初始化是否完成
		Mach_Control.An_b.An_GohomeHMI:=FALSE;
		Mach_Control.Ca_b.Ca_GohomeHMI:=FALSE;
		IF Mach_Control.Ca_b.Ca_GohomeDone AND Mach_Control.An_b.An_GohomeDone AND 
		 arrAxisCtrl[AxiseNo.AxisName.AnDTCarryingLine].Cmd.arrbRealPoint[1] AND arrAxisCtrl[AxiseNo.AxisName.CaDTCarryingLine].Cmd.arrbRealPoint[1] THEN
				Mach_Control.DT_b.Step[0]:=30;
		END_IF
30://叠台部分初始化
		Mach_Control.DT_b.DTIniti_Hbtn:=TRUE;
		Mach_Control.DT_b.Step[0]:=40;
40://判断叠台初始化是否完成
	Mach_Control.DT_b.DTIniti_Hbtn:=FALSE;
	IF Mach_Control.DT_b.DTIniti_Done THEN							
		Mach_Control.DT_b.Step[0]:=0;
	END_IF	
END_CASE
IF Step_InitCaDT=9999 OR Step_InitAnDT=9999 OR Step_InitDT=9999 THEN
	Mach_Control.DT_b.Step[0]:=0;
END_IF
			
			
(*********************************************************************************叠台部分轴回原点********************************************************************************************)		
//判断叠台是否回原点完成
IF arrAxisCtrl[AxiseNo.AxisName.SEPTATCache].Status.Homed AND arrAxisCtrl[AxiseNo.AxisName.SEPTAdeviation1].Status.Homed AND arrAxisCtrl[AxiseNo.AxisName.SEPTAdeviation2].Status.Homed AND
	arrAxisCtrl[AxiseNo.AxisName.LeftYDUpDown].Status.Homed AND arrAxisCtrl[AxiseNo.AxisName.LeftYDLine].Status.Homed AND arrAxisCtrl[AxiseNo.AxisName.RightYDUpDown].Status.Homed AND
	arrAxisCtrl[AxiseNo.AxisName.RightYDLine].Status.Homed AND arrAxisCtrl[AxiseNo.AxisName.SEPTATLine].Status.Homed AND DTIniti_Done THEN
	Mach_Control.DT_b.DTIniti_Done:=TRUE;//叠台回原点完成
ELSE
	Mach_Control.DT_b.DTIniti_Done:=FALSE;//叠台回原点完成
END_IF


	
	CASE Step_InitDT OF 		
			0://等待叠台初始化启动
				IF fDT_GohmeTRGI.Q AND arrAxisCtrl[AxiseNo.AxisName.AnDTCarryingLine].Cmd.arrbRealPoint[1] AND arrAxisCtrl[AxiseNo.AxisName.CaDTCarryingLine].Cmd.arrbRealPoint[1]  THEN
					Dietai_GohomeDone:=FALSE;//叠台回原点完成
		           		Dietai_Gohoming:=TRUE;//叠台回原点中
					Mach_Control.DT_b.DTIniti_Hbtn:=FALSE;
					Step_InitDT:=1;
				END_IF
			1://复位回原点完成
					DTIniti_Done:=FALSE;//叠台回原点完成
					tDT_GohomeTON.IN:=FALSE;
					IF NOT DTIniti_Done THEN
							Step_InitDT:=10;
					END_IF
			10://
				
				DP_Step0:=0;
				DP_Step1:=0;	
				DP_Step3:=0;
				DP_Step4:=0;
				DP_Step11:=0;
				DP_Step12:=0;
				iTensionAutoStep:=0;
				bFirstFoldFinish[1] R=Mach_Control.An_b.An_FirstFoldCnt=0 AND Mach_Control.Ca_b.Ca_FirstFoldCnt=0;//首层隔膜空叠
				bFirstFoldFinish[2]:=FALSE;//正常电芯空叠隔膜
				bFirstFoldFinish[3]:=FALSE;//接带、黄标空叠隔膜
				bEmptyFoldMark[1] R=Mach_Control.An_b.An_FirstFoldCnt=0 AND Mach_Control.Ca_b.Ca_FirstFoldCnt=0;//进入空叠流程
				bEmptyFoldMark[2]:=FALSE;//进入空叠流程
				bEmptyFoldMark[3]:=FALSE;//进入空叠流程	
				//Mach_Control.An_b.An_FirstFoldCnt:=0;
				//Mach_Control.Ca_b.Ca_FirstFoldCnt:=0;
				iEmptyFoldStep[1]:=0;
				iEmptyFoldStep[2]:=0;
				iEmptyFoldStep[3]:=0;
				Mach_Control.An_b.An_KDQuantited :=0;
				Mach_Control.Ca_b.Ca_KDQuantited:=0;
				Mach_Control.DT_b.OverhandFirstPice:=0;
				Ca_OverNGStep:=0;	
				An_OverNGStep:=0;								
	        	An_OverNGMark:=FALSE;	
	        	Ca_OverNGMark:=FALSE;
				OversequelNG:=FALSE;	
	
				DT_Readydown:=FALSE;
				DP_CheseCam:=FALSE;	
				CellMemory[Mach_Control.DT_b.DT_Memory].Cell:=FALSE;	
				Mach_Control.DT_b.OffloadRequest:=FALSE;//叠电芯完成，请求下电芯
				CellMemory[Mach_Control.DT_b.DT_Memory].Overhang_TF:=FALSE;	//叠电芯对齐度NG踢废信号
				Mach_Control.DT_b.Overhang_TF:=FALSE;
				
				arrCyCtrl[arrCyNo.CylinderName.PoleInflationCy].Cmd.bON:=TRUE;
				fbCamInLeftYDLine.bCamInExecute:=FALSE;//左压刀开合
				fbCamInLeftYDUpDown.bCamInExecute:=FALSE;//左压刀升降
				fbCamInRightYDLine.bCamInExecute:=FALSE;//右压刀开合
				fbCamInRightYDUpDown.bCamInExecute:=FALSE;//左压刀升降
				
				fbCamInGMBuffer.bCamInExecute:=FALSE;//隔膜缓存
				fbCamInGMDanserMove.bCamInExecute:=FALSE;//隔膜平移
				fbCamInVirGMDriver.bCamInExecute:=FALSE;//隔膜放卷虚轴
				
               	 		arrCyCtrl[arrCyNo.CylinderName.PreDiaph].Cmd.bOFF:=TRUE;//叠台压隔膜气缸缩回	
				VirMain_TON.IN:=FALSE;
				arrAxisCtrl[AxiseNo.VirAxisName.VirMain].Cmd	.bMoveAbs:=FALSE;	
				IF arrCyCtrl[arrCyNo.CylinderName.PreDiaph].Io.DIOFFSwitch AND NOT fbCamInLeftYDLine.bCamInExecute AND 
					NOT fbCamInLeftYDUpDown.bCamInExecute AND NOT fbCamInRightYDLine.bCamInExecute AND 
					NOT  fbCamInRightYDUpDown.bCamInExecute AND NOT fbCamInGMBuffer.bCamInExecute AND 
					NOT fbCamInGMDanserMove.bCamInExecute AND NOT fbCamInVirGMDriver.bCamInExecute  THEN
					 
						Step_InitDT:=20;
				END_IF	
			20://轴停止 
				arrAxisCtrl[AxiseNo.AxisName.SEPTATCache].Cmd.bHalt:=TRUE;//隔膜缓存解耦
				arrAxisCtrl[AxiseNo.AxisName.SEPTAdeviation1].Cmd.bHalt:=TRUE;//隔膜放卷纠偏解耦
				arrAxisCtrl[AxiseNo.AxisName.SEPTAdeviation2].Cmd.bHalt:=TRUE;//隔膜尾部纠偏解耦
				arrAxisCtrl[AxiseNo.AxisName.LeftYDUpDown].Cmd.bHalt:=TRUE;//左压刀升降轴解耦
				arrAxisCtrl[AxiseNo.AxisName.LeftYDLine].Cmd.bHalt:=TRUE;//左压刀开合轴解耦
				arrAxisCtrl[AxiseNo.AxisName.RightYDUpDown].Cmd.bHalt:=TRUE;//右压刀升降轴解耦
				arrAxisCtrl[AxiseNo.AxisName.RightYDLine].Cmd.bHalt:=TRUE;//右压刀开合轴解耦
				arrAxisCtrl[AxiseNo.AxisName.SEPTATLine].Cmd.bHalt:=TRUE;//隔膜平移轴解耦			
				 IF  	NOT arrAxisCtrl[AxiseNo.AxisName.SEPTATCache].Status.Coupled AND arrAxisCtrl[AxiseNo.AxisName.SEPTATCache].Status.NoMoving AND
					   NOT arrAxisCtrl[AxiseNo.AxisName.SEPTAdeviation1].Status.Coupled AND arrAxisCtrl[AxiseNo.AxisName.SEPTAdeviation1].Status.NoMoving AND
					   NOT arrAxisCtrl[AxiseNo.AxisName.SEPTAdeviation2].Status.Coupled AND arrAxisCtrl[AxiseNo.AxisName.SEPTAdeviation2].Status.NoMoving AND 
					   NOT arrAxisCtrl[AxiseNo.AxisName.LeftYDUpDown].Status.Coupled AND arrAxisCtrl[AxiseNo.AxisName.LeftYDUpDown].Status.NoMoving AND
					   NOT arrAxisCtrl[AxiseNo.AxisName.LeftYDLine].Status.Coupled AND arrAxisCtrl[AxiseNo.AxisName.LeftYDLine].Status.NoMoving AND
					   NOT arrAxisCtrl[AxiseNo.AxisName.RightYDUpDown].Status.Coupled AND arrAxisCtrl[AxiseNo.AxisName.RightYDUpDown].Status.NoMoving AND
					   NOT arrAxisCtrl[AxiseNo.AxisName.RightYDLine].Status.Coupled AND arrAxisCtrl[AxiseNo.AxisName.RightYDLine].Status.NoMoving AND
					   NOT arrAxisCtrl[AxiseNo.AxisName.SEPTATLine].Status.Coupled AND	arrAxisCtrl[AxiseNo.AxisName.SEPTATLine].Status.NoMoving THEN
							arrAxisCtrl[AxiseNo.AxisName.SEPTATCache].Cmd.bHalt:=FALSE;//隔膜缓存解耦
							arrAxisCtrl[AxiseNo.AxisName.SEPTAdeviation1].Cmd.bHalt:=FALSE;//隔膜放卷纠偏解耦
							arrAxisCtrl[AxiseNo.AxisName.SEPTAdeviation2].Cmd.bHalt:=FALSE;//隔膜尾部纠偏解耦
							arrAxisCtrl[AxiseNo.AxisName.LeftYDUpDown].Cmd.bHalt:=FALSE;//左压刀升降轴解耦
							arrAxisCtrl[AxiseNo.AxisName.LeftYDLine].Cmd.bHalt:=FALSE;//左压刀开合轴解耦
							arrAxisCtrl[AxiseNo.AxisName.RightYDUpDown].Cmd.bHalt:=FALSE;//右压刀升降轴解耦
							arrAxisCtrl[AxiseNo.AxisName.RightYDLine].Cmd.bHalt:=FALSE;//右压刀开合轴解耦
							arrAxisCtrl[AxiseNo.AxisName.SEPTATLine].Cmd.bHalt:=FALSE;//隔膜平移轴解耦										   							   
							Step_InitDT:=30;
				   END_IF				   
				30://轴上使能
						arrAxisCtrl[AxiseNo.AxisName.SEPTATCache].Cmd.bEnable:=TRUE;//隔膜缓存
						arrAxisCtrl[AxiseNo.AxisName.SEPTAdeviation1].Cmd.bEnable:=TRUE;//隔膜放卷纠偏
						arrAxisCtrl[AxiseNo.AxisName.SEPTAdeviation2].Cmd.bEnable:=TRUE;//隔膜尾部纠偏
						arrAxisCtrl[AxiseNo.AxisName.LeftYDUpDown].Cmd.bEnable:=TRUE;//左压刀升降轴
						arrAxisCtrl[AxiseNo.AxisName.LeftYDLine].Cmd.bEnable:=TRUE;//左压刀开合轴
						arrAxisCtrl[AxiseNo.AxisName.RightYDUpDown].Cmd.bEnable:=TRUE;//右压刀升降轴
						arrAxisCtrl[AxiseNo.AxisName.RightYDLine].Cmd.bEnable:=TRUE;//右压刀开合轴
						arrAxisCtrl[AxiseNo.AxisName.SEPTATLine].Cmd.bEnable:=TRUE;//隔膜平移轴		
						 IF  arrAxisCtrl[AxiseNo.AxisName.SEPTATCache].Status.Enabled AND 
							   arrAxisCtrl[AxiseNo.AxisName.SEPTAdeviation1].Status.Enabled AND 
							   arrAxisCtrl[AxiseNo.AxisName.SEPTAdeviation2].Status.Enabled AND 
							   arrAxisCtrl[AxiseNo.AxisName.LeftYDUpDown].Status.Enabled AND 
							   arrAxisCtrl[AxiseNo.AxisName.LeftYDLine].Status.Enabled AND 
							   arrAxisCtrl[AxiseNo.AxisName.RightYDUpDown].Status.Enabled AND 
							   arrAxisCtrl[AxiseNo.AxisName.RightYDLine].Status.Enabled AND 
							   arrAxisCtrl[AxiseNo.AxisName.SEPTATLine].Status.Enabled THEN
							Step_InitDT:=40;
						ELSIF    arrAxisCtrl[AxiseNo.AxisName.SEPTATCache].Status.Error OR 
								   arrAxisCtrl[AxiseNo.AxisName.SEPTAdeviation1].Status.Error OR 
								   arrAxisCtrl[AxiseNo.AxisName.SEPTAdeviation2].Status.Error OR 
								   arrAxisCtrl[AxiseNo.AxisName.LeftYDUpDown].Status.Error OR 
								   arrAxisCtrl[AxiseNo.AxisName.LeftYDLine].Status.Error OR 
								   arrAxisCtrl[AxiseNo.AxisName.RightYDUpDown].Status.Error OR 
								   arrAxisCtrl[AxiseNo.AxisName.RightYDLine].Status.Error OR 
								   arrAxisCtrl[AxiseNo.AxisName.SEPTATLine].Status.Error THEN
							Dietai_Gohoming:=FALSE;//叠台回原点中	   
							Step_InitDT:=9999;								
						END_IF	   
			40://隔膜缓存回原点、隔膜纠偏上回原点、隔膜纠偏下回原点
				
				arrAxisCtrl[AxiseNo.AxisName.SEPTATCache].Cmd.bHome:=TRUE;//隔膜缓存回原点
				arrAxisCtrl[AxiseNo.AxisName.SEPTAdeviation1].Cmd.bHome:=TRUE;//隔膜放卷纠偏回原点
				arrAxisCtrl[AxiseNo.AxisName.SEPTAdeviation2].Cmd.bHome:=TRUE;//隔膜尾部纠偏回原点
				Step_InitDT:=50;
			50://判断轴回原点是否完成
				  IF NOT tDT_GohomeTON.Q THEN
							  tDT_GohomeTON.IN:=TRUE;
				  ELSE
					  IF arrAxisCtrl[AxiseNo.AxisName.SEPTATCache].Status.Homed AND arrAxisCtrl[AxiseNo.AxisName.SEPTATCache].Status.NoMoving AND
						  arrAxisCtrl[AxiseNo.AxisName.SEPTAdeviation1].Status.Homed AND arrAxisCtrl[AxiseNo.AxisName.SEPTAdeviation1].Status.NoMoving AND 
						  arrAxisCtrl[AxiseNo.AxisName.SEPTAdeviation2].Status.Homed AND arrAxisCtrl[AxiseNo.AxisName.SEPTAdeviation2].Status.NoMoving THEN
						  tDT_GohomeTON.IN:=FALSE;
						  arrAxisCtrl[AxiseNo.AxisName.SEPTATCache].Cmd.bHome:=FALSE;//隔膜缓存回原点
						  arrAxisCtrl[AxiseNo.AxisName.SEPTAdeviation1].Cmd.bHome:=FALSE;//隔膜放卷纠偏回原点
						  arrAxisCtrl[AxiseNo.AxisName.SEPTAdeviation2].Cmd.bHome:=FALSE;//隔膜尾部纠偏回原点
						  Step_InitDT:=51;
						ELSIF arrAxisCtrl[AxiseNo.AxisName.SEPTATCache].Status.Error OR  arrAxisCtrl[AxiseNo.AxisName.SEPTAdeviation1].Status.Error OR 
							arrAxisCtrl[AxiseNo.AxisName.SEPTAdeviation2].Status.Error THEN
							tDT_GohomeTON.IN:=FALSE;
							arrAxisCtrl[AxiseNo.AxisName.SEPTATCache].Cmd.bHome:=FALSE;//隔膜缓存回原点
							arrAxisCtrl[AxiseNo.AxisName.SEPTAdeviation1].Cmd.bHome:=FALSE;//隔膜放卷纠偏回原点
							arrAxisCtrl[AxiseNo.AxisName.SEPTAdeviation2].Cmd.bHome:=FALSE;//隔膜尾部纠偏回原点
							Dietai_Gohoming:=FALSE;//叠台回原点中
							Step_InitDT:=9999;											 
					  END_IF
				  END_IF
			51://缓存、放卷纠偏、底部纠偏
				  IF NOT tDT_GohomeTON.Q THEN
				  	tDT_GohomeTON.IN:=TRUE;		
				  ELSE	
								IF NOT arrAxisCtrl[AxiseNo.AxisName.SEPTATCache].Cmd.arrbRealPoint[1] AND  arrAxisCtrl[AxiseNo.AxisName.SEPTATCache].Status.NoMoving THEN
								   arrAxisCtrl[AxiseNo.AxisName.SEPTATCache].Cmd.iGoSetPos:=1;
								END_IF					
								IF NOT arrAxisCtrl[AxiseNo.AxisName.SEPTAdeviation1].Cmd.arrbRealPoint[1] AND  arrAxisCtrl[AxiseNo.AxisName.SEPTAdeviation1].Status.NoMoving THEN
								   arrAxisCtrl[AxiseNo.AxisName.SEPTAdeviation1].Cmd.iGoSetPos:=1;
								END_IF	
								IF NOT arrAxisCtrl[AxiseNo.AxisName.SEPTAdeviation2].Cmd.arrbRealPoint[1] AND  arrAxisCtrl[AxiseNo.AxisName.SEPTAdeviation2].Status.NoMoving THEN
								   arrAxisCtrl[AxiseNo.AxisName.SEPTAdeviation2].Cmd.iGoSetPos:=1;
								END_IF			
								IF   arrAxisCtrl[AxiseNo.AxisName.SEPTATCache].Cmd.arrbRealPoint[1]  AND arrAxisCtrl[AxiseNo.AxisName.SEPTAdeviation1].Cmd.arrbRealPoint[1] AND 
									  arrAxisCtrl[AxiseNo.AxisName.SEPTAdeviation2].Cmd.arrbRealPoint[1] THEN
									  	tDT_GohomeTON.IN:=FALSE;	
										Step_InitDT:=55;
								ELSIF arrAxisCtrl[AxiseNo.AxisName.SEPTATCache].Status.Error OR arrAxisCtrl[AxiseNo.AxisName.SEPTAdeviation1].Status.Error OR arrAxisCtrl[AxiseNo.AxisName.SEPTAdeviation2].Status.Error THEN
										tDT_GohomeTON.IN:=FALSE;	
										Dietai_Gohoming:=FALSE;//叠台回原点中
										Step_InitDT:=9999;
								END_IF
					END_IF
					
			55://判断左右压刀开合、升降是否在初始位,与其都已经回原完成
				IF 	arrAxisCtrl[AxiseNo.AxisName.LeftYDLine].Cmd.arrbRealPoint[1] AND arrAxisCtrl[AxiseNo.AxisName.LeftYDLine].Status.Homed AND 
					arrAxisCtrl[AxiseNo.AxisName.LeftYDUpDown].Cmd.arrbRealPoint[1] AND arrAxisCtrl[AxiseNo.AxisName.LeftYDUpDown].Status.Homed AND
					arrAxisCtrl[AxiseNo.AxisName.RightYDLine].Cmd.arrbRealPoint[1] AND arrAxisCtrl[AxiseNo.AxisName.RightYDLine].Status.Homed AND
					arrAxisCtrl[AxiseNo.AxisName.RightYDUpDown].Cmd.arrbRealPoint[1] AND arrAxisCtrl[AxiseNo.AxisName.RightYDUpDown].Status.Homed THEN
					Step_InitDT:=180;
					ELSE
					Step_InitDT:=60;	
				END_IF
				
					
		
			60://左压刀升降轴回原点
				arrAxisCtrl[AxiseNo.AxisName.LeftYDUpDown].Cmd.bHome:=TRUE;//左压刀升降轴回原点
				Step_InitDT:=70;
			70://判断左压刀升降轴回原是否完成
				  IF NOT tDT_GohomeTON.Q THEN
							  tDT_GohomeTON.IN:=TRUE;
				  ELSE
							  IF arrAxisCtrl[AxiseNo.AxisName.LeftYDUpDown].Status.Homed AND arrAxisCtrl[AxiseNo.AxisName.LeftYDUpDown].Status.NoMoving THEN
									arrAxisCtrl[AxiseNo.AxisName.LeftYDUpDown].Cmd.bHome:=FALSE;//左压刀升降轴回原点
									tDT_GohomeTON.IN:=FALSE;
								  	Step_InitDT:=80;
							  ELSIF arrAxisCtrl[AxiseNo.AxisName.LeftYDUpDown].Status.Error THEN
								  	arrAxisCtrl[AxiseNo.AxisName.LeftYDUpDown].Cmd.bHome:=FALSE;//左压刀升降轴回原点
									tDT_GohomeTON.IN:=FALSE;
									Dietai_Gohoming:=FALSE;//叠台回原点中
								  	Step_InitDT:=9999;							  
							  END_IF
					END_IF		
					
			80://左压刀开合轴回原点
				arrCyCtrl[arrCyNo.ElectValveName.DTVacuum].Cmd.bON:=FALSE;
				arrCyCtrl[arrCyNo.ElectValveName.DTVacuum].Cmd.bOFF:=TRUE;
				arrAxisCtrl[AxiseNo.AxisName.LeftYDLine].Cmd.bHome:=TRUE;//左压刀开合轴回原点
				Step_InitDT:=90;
			90://判断左压刀开合轴回原点是否完成
				  IF NOT tDT_GohomeTON.Q THEN
							  tDT_GohomeTON.IN:=TRUE;
				  ELSE
						IF arrAxisCtrl[AxiseNo.AxisName.LeftYDLine].Status.Homed AND arrAxisCtrl[AxiseNo.AxisName.LeftYDLine].Status.NoMoving  THEN
							tDT_GohomeTON.IN:=FALSE;
							arrAxisCtrl[AxiseNo.AxisName.LeftYDLine].Cmd.bHome:=FALSE;//左压刀开合轴回原点
							Step_InitDT:=100;
						ELSIF arrAxisCtrl[AxiseNo.AxisName.LeftYDLine].Status.Error THEN
							tDT_GohomeTON.IN:=FALSE;
							arrAxisCtrl[AxiseNo.AxisName.LeftYDLine].Cmd.bHome:=FALSE;//左压刀开合轴回原点
							Dietai_Gohoming:=FALSE;//叠台回原点中
							Step_InitDT:=9999;
						END_IF
				END_IF
			100://左压刀开合轴移动至初始位
				IF NOT arrAxisCtrl[AxiseNo.AxisName.LeftYDLine].Cmd.arrbRealPoint[1] AND arrAxisCtrl[AxiseNo.AxisName.LeftYDLine].Status.NoMoving THEN//左压刀开合轴移动至初始位
				   arrAxisCtrl[AxiseNo.AxisName.LeftYDLine].Cmd.iGoSetPos:=1;
				END_IF
				IF arrAxisCtrl[AxiseNo.AxisName.LeftYDLine].Status.Error THEN
					Dietai_Gohoming:=FALSE;//叠台回原点中
					Step_InitDT:=9999;
				ELSIF arrAxisCtrl[AxiseNo.AxisName.LeftYDLine].Cmd.arrbRealPoint[1] AND arrAxisCtrl[AxiseNo.AxisName.LeftYDLine].Status.NoMoving THEN
					Step_InitDT:=110;
				END_IF
			110://左压刀升降轴移动至初始位
				IF NOT arrAxisCtrl[AxiseNo.AxisName.LeftYDUpDown].Cmd.arrbRealPoint[1] AND arrAxisCtrl[AxiseNo.AxisName.LeftYDUpDown].Status.NoMoving  THEN//左压刀开合轴移动至初始位
				   arrAxisCtrl[AxiseNo.AxisName.LeftYDUpDown].Cmd.iGoSetPos:=1;
				END_IF
				IF arrAxisCtrl[AxiseNo.AxisName.LeftYDUpDown].Status.Error THEN
					Dietai_Gohoming:=FALSE;//叠台回原点中
					Step_InitDT:=9999;
				ELSIF arrAxisCtrl[AxiseNo.AxisName.LeftYDUpDown].Cmd.arrbRealPoint[1] AND arrAxisCtrl[AxiseNo.AxisName.LeftYDUpDown].Status.NoMoving THEN
					Step_InitDT:=120;
				END_IF
			120://右压刀升降轴回原点
				arrAxisCtrl[AxiseNo.AxisName.RightYDUpDown].Cmd.bHome:=TRUE;//右压刀升降轴回原点
				Step_InitDT:=130;
			130://判断轴回原点是否完成
				  IF NOT tDT_GohomeTON.Q THEN
							  tDT_GohomeTON.IN:=TRUE;
				  ELSE
							IF  arrAxisCtrl[AxiseNo.AxisName.RightYDUpDown].Status.Homed AND arrAxisCtrl[AxiseNo.AxisName.RightYDUpDown].Status.NoMoving THEN
								tDT_GohomeTON.IN:=FALSE;
								arrAxisCtrl[AxiseNo.AxisName.RightYDUpDown].Cmd.bHome:=FALSE;//右压刀升降轴回原点
								Step_InitDT:=140;
							ELSIF arrAxisCtrl[AxiseNo.AxisName.RightYDUpDown].Status.Error THEN
									tDT_GohomeTON.IN:=FALSE;
									arrAxisCtrl[AxiseNo.AxisName.RightYDUpDown].Cmd.bHome:=FALSE;//右压刀升降轴回原点
									Dietai_Gohoming:=FALSE;//叠台回原点中
									Step_InitDT:=9999;
							END_IF	
				END_IF
			140://右压刀开合轴回原点
				arrAxisCtrl[AxiseNo.AxisName.RightYDLine].Cmd.bHome:=TRUE;//右压刀开合轴回原点
				Step_InitDT:=150;
			150://判断开合轴回原点是否完成
				  IF NOT tDT_GohomeTON.Q THEN
							  tDT_GohomeTON.IN:=TRUE;
				  ELSE
							  IF arrAxisCtrl[AxiseNo.AxisName.RightYDLine].Status.Homed AND arrAxisCtrl[AxiseNo.AxisName.RightYDLine].Status.NoMoving THEN
									 tDT_GohomeTON.IN:=FALSE;
									arrAxisCtrl[AxiseNo.AxisName.RightYDLine].Cmd.bHome:=FALSE;//右压刀开合轴回原点
									Step_InitDT:=160;
							   ELSIF arrAxisCtrl[AxiseNo.AxisName.RightYDLine].Status.Error THEN
								   		 tDT_GohomeTON.IN:=FALSE;
										arrAxisCtrl[AxiseNo.AxisName.RightYDLine].Cmd.bHome:=FALSE;//右压刀开合轴回原点
										Dietai_Gohoming:=FALSE;//叠台回原点中
										Step_InitDT:=9999;				   
							  END_IF	
					END_IF
			160://右压刀开合轴移动至初始位
				IF NOT arrAxisCtrl[AxiseNo.AxisName.RightYDLine].Cmd.arrbRealPoint[1] AND arrAxisCtrl[AxiseNo.AxisName.RightYDLine].Status.NoMoving THEN//右压刀开合轴移动至初始位
				   arrAxisCtrl[AxiseNo.AxisName.RightYDLine].Cmd.iGoSetPos:=1;
				END_IF
				IF arrAxisCtrl[AxiseNo.AxisName.RightYDLine].Status.Error THEN
					Dietai_Gohoming:=FALSE;//叠台回原点中
					Step_InitDT:=9999;
				ELSIF arrAxisCtrl[AxiseNo.AxisName.RightYDLine].Cmd.arrbRealPoint[1] AND arrAxisCtrl[AxiseNo.AxisName.RightYDLine].Status.NoMoving THEN
					Step_InitDT:=170;
				END_IF	
			170://右压刀升降轴移动至初始位	
				IF NOT arrAxisCtrl[AxiseNo.AxisName.RightYDUpDown].Cmd.arrbRealPoint[1] AND arrAxisCtrl[AxiseNo.AxisName.RightYDUpDown].Status.NoMoving THEN//右压刀升降轴移动至初 始位
				   arrAxisCtrl[AxiseNo.AxisName.RightYDUpDown].Cmd.iGoSetPos:=1;
				END_IF
				IF arrAxisCtrl[AxiseNo.AxisName.RightYDUpDown].Status.Error THEN
					Dietai_Gohoming:=FALSE;//叠台回原点中
					Step_InitDT:=9999;
				ELSIF arrAxisCtrl[AxiseNo.AxisName.RightYDUpDown].Cmd.arrbRealPoint[1] AND arrAxisCtrl[AxiseNo.AxisName.RightYDUpDown].Status.NoMoving  THEN
					Step_InitDT:=180;
				END_IF	
			180://隔膜平移轴回原点
				IF arrAxisCtrl[AxiseNo.AxisName.AnDTCarryingLine].Cmd.arrbRealPoint[1] AND arrAxisCtrl[AxiseNo.AxisName.CaDTCarryingLine].Cmd.arrbRealPoint[1] 
					AND arrAxisCtrl[AxiseNo.AxisName.LeftYDLine].Cmd.arrbRealPoint[1] AND arrAxisCtrl[AxiseNo.AxisName.LeftYDLine].Status.Homed AND 
					arrAxisCtrl[AxiseNo.AxisName.LeftYDUpDown].Cmd.arrbRealPoint[1] AND arrAxisCtrl[AxiseNo.AxisName.LeftYDUpDown].Status.Homed AND
					arrAxisCtrl[AxiseNo.AxisName.RightYDLine].Cmd.arrbRealPoint[1] AND arrAxisCtrl[AxiseNo.AxisName.RightYDLine].Status.Homed AND
					arrAxisCtrl[AxiseNo.AxisName.RightYDUpDown].Cmd.arrbRealPoint[1] AND arrAxisCtrl[AxiseNo.AxisName.RightYDUpDown].Status.Homed  THEN
						arrAxisCtrl[AxiseNo.AxisName.SEPTATLine].Cmd.bHome:=TRUE;//隔膜平移轴回原点
						Step_InitDT:=190;
				END_IF	
			190://判断回原点是否完成
				  IF NOT tDT_GohomeTON.Q THEN
							  tDT_GohomeTON.IN:=TRUE;
				  ELSE
						IF 	arrAxisCtrl[AxiseNo.AxisName.SEPTATLine].Status.Homed THEN
							 tDT_GohomeTON.IN:=FALSE;
							arrAxisCtrl[AxiseNo.AxisName.SEPTATLine].Cmd.bHome:=FALSE;//隔膜平移轴回原点
							Step_InitDT:=200;
						ELSIF arrAxisCtrl[AxiseNo.AxisName.SEPTATLine].Status.Error THEN
							tDT_GohomeTON.IN:=FALSE;
							arrAxisCtrl[AxiseNo.AxisName.SEPTATLine].Cmd.bHome:=FALSE;//隔膜平移轴回原点
							Dietai_Gohoming:=FALSE;//叠台回原点中
							Step_InitDT:=9999;
						END_IF	
					END_IF
			200://隔膜平移轴移动至初始位
				IF NOT arrAxisCtrl[AxiseNo.AxisName.SEPTATLine].Cmd.arrbRealPoint[1] AND  arrAxisCtrl[AxiseNo.AxisName.SEPTATLine].Status.NoMoving THEN//左压刀开合轴移动至初始位
				   arrAxisCtrl[AxiseNo.AxisName.SEPTATLine].Cmd.iGoSetPos:=1;
				END_IF
				IF NOT arrAxisCtrl[AxiseNo.AxisName.SEPTATCache].Cmd.arrbRealPoint[1] AND  arrAxisCtrl[AxiseNo.AxisName.SEPTATCache].Status.NoMoving THEN//左压刀开合轴移动至初始位
				   arrAxisCtrl[AxiseNo.AxisName.SEPTATCache].Cmd.iGoSetPos:=1;
				END_IF
				IF arrAxisCtrl[AxiseNo.AxisName.SEPTATLine].Cmd.arrbRealPoint[1] AND  arrAxisCtrl[AxiseNo.AxisName.SEPTATLine].Status.NoMoving AND 
					 arrAxisCtrl[AxiseNo.AxisName.SEPTATCache].Cmd.arrbRealPoint[1] AND  arrAxisCtrl[AxiseNo.AxisName.SEPTATCache].Status.NoMoving THEN
							DTIniti_Done:=TRUE;//叠台回原点完成
							Dietai_Gohoming:=FALSE;//叠台回原点中
							Dietai_GohomeDone:=TRUE;//叠台回原点完成
							Step_InitDT:=0;
				ELSIF arrAxisCtrl[AxiseNo.AxisName.SEPTATLine].Status.Error OR arrAxisCtrl[AxiseNo.AxisName.SEPTATCache].Status.Error THEN
					        Dietai_Gohoming:=FALSE;//叠台回原点中
							Step_InitDT:=9999;
				END_IF				
	END_CASE
END_IF
END_ACTION

ACTION DT_Alarm:
DT_AlarmTon[0](PT:=T#2S);
DT_AlarmTon[1](PT:=T#10MS);
DT_AlarmTon[2](PT:=T#100MS);
DT_AlarmTon[3](PT:=T#2S);
DT_AlarmTon[4](IN:=   NOT Mach_Control.DT_b.bTensionOK AND Mach_Control.U.DT_iMode=1  AND DP_Step0=0, PT:=T#60S , Q=> , ET=> );
//Mach_Control.DT_b.Error[1]:=TRUE;//隔膜缓存凸轮创建失败
//Mach_Control.DT_b.Error[2] :=TRUE;//叠台储气罐真空不足报警
//Mach_Control.DT_b.Error[3]:=TRUE;////凸轮耦合时，左压刀升降不在低位
//Mach_Control.DT_b.Error[4]:=TRUE;//凸轮耦合时，右压刀升降不在低位
//Mach_Control.DT_b.Error[5]:=TRUE;//叠负极片凸轮耦合时，隔膜平移轴即不在负极叠片位，也不在正极叠片位报警
//Mach_Control.DT_b.Error[6]:=TRUE;//叠正极片凸轮耦合时，隔膜平移轴即不在负极叠片位，也不在正极叠片位报警
//Mach_Control.DT_b.Error[7]:=TRUE;//叠正极片凸轮耦合时，负极取片即不在取片位，也不在叠片位
//Mach_Control.DT_b.Error[8]:=TRUE;//叠正极片凸轮耦合时，正极片不在取片位
//Mach_Control.DT_b.Error[9];//纠偏凸轮耦合失败报警
//Mach_Control.DT_b.Error[10];//纠偏左限位报警
//Mach_Control.DT_b.Error[11];//纠偏右限位报警
//Mach_Control.DT_b.Error[12]=左压刀开合凸轮耦合报警
//Mach_Control.DT_b.Error[13]=左压刀升降凸轮耦合报警
//Mach_Control.DT_b.Error[14]=右压刀开合凸轮耦合报警
//Mach_Control.DT_b.Error[15]=右压刀升降凸轮耦合报警
//Mach_Control.DT_b.Error[16]=隔膜放卷凸轮报警
//Mach_Control.DT_b.Error[17]=隔膜平移凸轮报警
//Mach_Control.DT_b.Error[18]=隔膜缓存凸轮报警
//Mach_Control.DT_b.Error[19]=凸轮耦合报警
//Mach_Control.DT_b.Error[20]:=TRUE;//CCD通讯异常
//Mach_Control.DT_b.Error[21];//隔膜纠偏报警
//Mach_Control.DT_b.Error[22]=主轴启动超时报警
//Mach_Control.DT_b.Error[23]=叠台回原点超时报警  
//Mach_Control.DT_b.Error[24] :=TRUE;//放卷卷径报警
//Mach_Control.DT_b.Error[25] :=TRUE;//正极已叠片数大于负极已叠片数报警
//Mach_Control.DT_b.Error[26] :=TRUE;//连续对齐度NG报警
//Mach_Control.DT_b.Error[27]:=TRUE;//检测到叠台重片，请查看是否重片
//Mach_Control.DT_b.Error[28] :=TRUE;//叠台左压刀使用已经超出寿命报警
//Mach_Control.DT_b.Error[29] :=TRUE;//叠台右压刀使用已经超出寿命报警
//Mach_Control.DT_b.Error[30];//凸轮耦合时，正极送片搬运平移不在取片位
//Mach_Control.DT_b.Error[31];凸轮耦合时，正极送片搬运平移不在放片位
//Mach_Control.DT_b.Error[32];凸轮耦合时，正极叠片搬运平移不在取片位
//Mach_Control.DT_b.Error[33];凸轮耦合时，正极叠片搬运平移不在放片位
//Mach_Control.DT_b.Error[34];凸轮耦合时，正极送片搬运旋转不在取片位
//Mach_Control.DT_b.Error[35];凸轮耦合时，正极送片搬运旋转不在放片位
//Mach_Control.DT_b.Error[36];凸轮耦合时，正极送片搬运升降不在等待高度
//Mach_Control.DT_b.Error[37];凸轮耦合时，正极叠片搬运升降不在等待高度  
//Mach_Control.DT_b.Error[38];//凸轮耦合时，负极送片搬运平移2不在取片位
//Mach_Control.DT_b.Error[39];//凸轮耦合时，负极送片搬运平移2不在放片位
//Mach_Control.DT_b.Error[40];//凸轮耦合时，负极叠片搬运平移不在取片位
//Mach_Control.DT_b.Error[41];//凸轮耦合时，负极叠片搬运平移不在放片位
//Mach_Control.DT_b.Error[42];//凸轮耦合时，负极送片搬运升降不在等待高度
//Mach_Control.DT_b.Error[43];//凸轮耦合时，负极叠片搬运升降不在等待高度  
//Mach_Control.DT_b.Error[44]:=TRUE;//自动时，隔膜气胀轴未涨紧报警		
//Mach_Control.DT_b.Error[45]////隔膜张力报警
//Mach_Control.DT_b.Error[46]=对齐度NG料盒料满
//Mach_Control.DT_b.Error[47]=对齐度NG剔废一次
//Mach_Control.DT_b.Error[48]=CCD工控机磁盘容量报警
//Mach_Control.DT_b.Error[49]=叠片平台当前极片折角报警
//Mach_Control.DT_b.Error[50]=触发对其度拍照时压刀在极片上面报警
//Mach_Control.DT_b.Error[51]=检测负极纠偏平台空片结果返回超时
//Mach_Control.DT_b.Error[52]=检测正极纠偏平台空片结果返回超时
//Mach_Control.DT_b.Error[53]=隔膜长度小于多少米
//Mach_Control.DT_b.Error[54]=陶瓷面感应器报警，请检查隔膜是否正确安装陶瓷面
//Mach_Control.DT_b.Error[55]叠首层隔膜过程中，隔膜平移轴未动作
//Mach_Control.DT_b.Error[56]叠台已到达清洁时间
//Mach_Control.DT_b.Error[57]空叠隔膜时正负极都不在取片位
//Mach_Control.DT_b.Error[58]---备用
//Mach_Control.DT_b.Error[59]叠台对齐度检测NG报警
//Mach_Control.DT_b.Error[60];//主轴启动前轴有故障
//Mach_Control.DT_b.Error[61];//主剩余隔膜不能叠一个电芯，请更换隔膜
//Mach_Control.DT_b.Error[62];//自动时隔膜张力未OK
//Mach_Control.DT_b.Error[63];//功能开关状态报警
//Mach_Control.DT_b.Error[64];//叠台有功能屏蔽报警
//Mach_Control.DT_b.Error[65];//压刀间距报警
//Mach_Control.DT_b.Error[66];//压刀铁氟龙计数到达设定值
//Mach_Control.DT_b.Error[67];//上电后叠台参数读取失败，请手动点读取参数
//Mach_Control.DT_b.Error[68];//正极对齐度拍照发送层数错误
//Mach_Control.DT_b.Error[69];//负极对齐度拍照发送层数错误
//Mach_Control.DT_b.Error[70];//正极对齐度接收结果为0
//Mach_Control.DT_b.Error[71];//负极对齐度接收结果为0
//叠台对齐度检测报警
IF Mach_Control.DT_b.iOverError=2 AND NOT Mach_Control.DT_b.DT_Overhang THEN
	//Mach_Control.DT_b.Error[59]:=TRUE;//对齐度检测
	Mach_Control.DT_b.Error_tips[6]:=TRUE;//叠台对齐度检测均值超限警告
END_IF
IF Mach_Control.DT_b.Error_tips[6]  AND fDT_AlarmRest.Q THEN
	Mach_Control.DT_b.iOverError:=0;
	Mach_Control.DT_b.Error_tips[6]:=FALSE;
END_IF
//对齐度连续超限检测预警
IF CCD.Over.Finish.OverhangXY_Warm=1 THEN
	Mach_Control.DT_b.Overhang_Warm:=TRUE;
(*ELSE
	CCD.Over.Start.OverhangXY_Warm_Reset:=1;*)
END_IF
IF Mach_Control.DT_b.Overhang_Warm AND Mach_Control.DT_b.Overhang_Warm_Reset THEN
	//CCD.Over.Start.OverhangXY_Warm_Reset:=0;
	CCD.Over.Finish.OverhangXY_Warm:=0;
	Mach_Control.DT_b.Overhang_Warm:=FALSE;
END_IF



IF    Mach_Control.se.Ceramics THEN//Mach_Control.U.DT_iMode=1 AND
	Mach_Control.DT_b.Error[54]:=TRUE;//陶瓷面感应器报警，请检查隔膜是否正确安装陶瓷面
//ELSE
//	Mach_Control.DT_b.Error[54]:=FALSE;//陶瓷面感应器报警，请检查隔膜是否正确安装陶瓷面
END_IF
IF  Par.stDT_date.CleanTimeHMIHour = System.StTime.wHour AND Par.stDT_date.CleanTimeHMIMin =System.stTime.wMinute THEN
	Mach_Control.DT_b.Error[56]:=TRUE;//请清洁机台叠台部分
END_IF

//清记录的标志位
IF rDT_AlarmRest.Q THEN
	FOR i:=1 TO 10 DO
		AnPosError[i] :=FALSE;
		CaPosError[i] :=FALSE;
		DTPosError[i] :=FALSE;
	END_FOR
END_IF
(********************************************************叠片时正负极搬运不在耦合位报警*****************************************************)
IF DP_Step0=9993 OR An_StandbyStep1=9993 OR Ca_StandbyStep0=9993 OR  DTPosError[11] THEN
 //正极取片轴不在耦合位报警	
 		PosErrorMark:=TRUE;//凸轮耦合时，有轴不在耦合位报警
   		IF arrAxisCtrl[AxiseNo.AxisName.AnDTCarryingLine].Cmd.arrbRealPoint[1] THEN
			   IF NOT arrAxisCtrl[AxiseNo.AxisName.AnCarryingLine].Cmd.arrbRealPoint[1]  THEN              
						Mach_Control.DT_b.Error[30]:=TRUE;//凸轮耦合时，正极送片搬运平移不在取片位
			   END_IF       		
		ELSIF arrAxisCtrl[AxiseNo.AxisName.AnDTCarryingLine].Cmd.arrbRealPoint[2] THEN
			   IF NOT arrAxisCtrl[AxiseNo.AxisName.AnCarryingLine].Cmd.arrbRealPoint[2] THEN             
				 	 Mach_Control.DT_b.Error[31]:=TRUE;//凸轮耦合时，正极送片搬运平移不在放片位
			   END_IF		   	   
        END_IF
		
		IF arrAxisCtrl[AxiseNo.AxisName.AnCarryingLine].Cmd.arrbRealPoint[1] THEN
			   IF NOT arrAxisCtrl[AxiseNo.AxisName.AnDTCarryingLine].Cmd.arrbRealPoint[1]  THEN              
				  	Mach_Control.DT_b.Error[32]:=TRUE;//凸轮耦合时，正极叠片搬运平移不在取片位
			   END_IF       		
		ELSIF arrAxisCtrl[AxiseNo.AxisName.AnCarryingLine].Cmd.arrbRealPoint[2] THEN
			   IF NOT arrAxisCtrl[AxiseNo.AxisName.AnDTCarryingLine].Cmd.arrbRealPoint[2] THEN             
				 	Mach_Control.DT_b.Error[33]:=TRUE;//凸轮耦合时，正极叠片搬运平移不在放片位
			   END_IF		   	   		   		   
        END_IF
		
		IF arrAxisCtrl[AxiseNo.AxisName.AnCarryingLine].Cmd.arrbRealPoint[1] THEN
			   IF NOT arrAxisCtrl[AxiseNo.AxisName.AnCarryingWhirling].Cmd.arrbRealPoint[1]  THEN             
						Mach_Control.DT_b.Error[34]:=TRUE;//凸轮耦合时，正极送片搬运旋转不在取片位
			   END_IF		
		ELSIF arrAxisCtrl[AxiseNo.AxisName.AnCarryingLine].Cmd.arrbRealPoint[2] THEN
			   IF NOT arrAxisCtrl[AxiseNo.AxisName.AnCarryingWhirling].Cmd.arrbRealPoint[2] THEN             
				 		Mach_Control.DT_b.Error[35]:=TRUE;//凸轮耦合时，正极送片搬运旋转不在放片位
			   END_IF
        END_IF

		IF NOT arrAxisCtrl[AxiseNo.AxisName.AnCarryingUpDown].Cmd.arrbRealPoint[4] THEN           
		 		Mach_Control.DT_b.Error[36]:=TRUE;//凸轮耦合时，正极送片搬运升降不在等待高度
	    END_IF  		   	
   
		IF NOT arrAxisCtrl[AxiseNo.AxisName.AnDTCarryingUpDown].Cmd.arrbRealPoint[4] THEN           
				Mach_Control.DT_b.Error[37]:=TRUE;//凸轮耦合时，正极叠片搬运升降不在等待高度  
	    END_IF 

		IF NOT arrAxisCtrl[AxiseNo.AxisName.LeftYDUpDown].Cmd.arrbRealPoint[1] THEN
				Mach_Control.DT_b.Error[3]:=TRUE;//凸轮耦合时，左压刀升降不在低位
		END_IF
		
		IF NOT arrAxisCtrl[AxiseNo.AxisName.RightYDUpDown].Cmd.arrbRealPoint[1] THEN
				Mach_Control.DT_b.Error[4]:=TRUE;//凸轮耦合时，右压刀升降不在低位
		END_IF
END_IF

IF DP_Step0=9994 OR An_StandbyStep1=9994 OR Ca_StandbyStep0=9994 OR  DTPosError[12]  THEN
//负极取片轴不在耦合位报警	
		PosErrorMark:=TRUE;//凸轮耦合时，有轴不在耦合位报警
   		IF arrAxisCtrl[AxiseNo.AxisName.CaDTCarryingLine].Cmd.arrbRealPoint[1] THEN
			   IF NOT arrAxisCtrl[AxiseNo.AxisName.CaCarryingLine2].Cmd.arrbRealPoint[1]  THEN             
						  Mach_Control.DT_b.Error[38]:=TRUE;//凸轮耦合时，负极送片搬运平移2不在取片位
			   END_IF		
		ELSIF arrAxisCtrl[AxiseNo.AxisName.CaDTCarryingLine].Cmd.arrbRealPoint[2] THEN
			   IF NOT arrAxisCtrl[AxiseNo.AxisName.CaCarryingLine2].Cmd.arrbRealPoint[2] THEN               
					  Mach_Control.DT_b.Error[39]:=TRUE;//凸轮耦合时，负极送片搬运平移2不在放片位
			   END_IF
        END_IF
		
		IF arrAxisCtrl[AxiseNo.AxisName.CaCarryingLine2].Cmd.arrbRealPoint[1] THEN
			   IF NOT arrAxisCtrl[AxiseNo.AxisName.CaDTCarryingLine].Cmd.arrbRealPoint[1]  THEN              
						Mach_Control.DT_b.Error[40]:=TRUE;//凸轮耦合时，负极叠片搬运平移不在取片位
			   END_IF		
		ELSIF arrAxisCtrl[AxiseNo.AxisName.CaCarryingLine2].Cmd.arrbRealPoint[2] THEN
			   IF NOT arrAxisCtrl[AxiseNo.AxisName.CaDTCarryingLine].Cmd.arrbRealPoint[2] THEN              
				 		Mach_Control.DT_b.Error[41]:=TRUE;//凸轮耦合时，负极叠片搬运平移不在放片位
			   END_IF
        END_IF
	
		IF NOT arrAxisCtrl[AxiseNo.AxisName.CaCarryingUpDown2].Cmd.arrbRealPoint[4] THEN            
		   		Mach_Control.DT_b.Error[42]:=TRUE;//凸轮耦合时，负极送片搬运升降不在等待高度
	    END_IF  		   	
   
		IF NOT arrAxisCtrl[AxiseNo.AxisName.CaDTCarryingUpDown].Cmd.arrbRealPoint[4] THEN          
		   		Mach_Control.DT_b.Error[43]:=TRUE;//凸轮耦合时，负极叠片搬运升降不在等待高度  
	    END_IF
	
		
		IF NOT arrAxisCtrl[AxiseNo.AxisName.LeftYDUpDown].Cmd.arrbRealPoint[1] THEN
				Mach_Control.DT_b.Error[3]:=TRUE;//凸轮耦合时，左压刀升降不在低位
		END_IF
		
		IF NOT arrAxisCtrl[AxiseNo.AxisName.RightYDUpDown].Cmd.arrbRealPoint[1] THEN
				Mach_Control.DT_b.Error[4]:=TRUE;//凸轮耦合时，右压刀升降不在低位
		END_IF  
END_IF


rDtUse[1](CLK:=PosErrorMark);

IF rDtUse[1].Q THEN
	PosErrorMark:=FALSE;//凸轮耦合时，有轴不在耦合位报警
	fActPos[1]:=arrAxisCtrl[AxiseNo.AxisName.AnCarryingLine].Status.fActPos;//正极送片搬运平移
	fSetPos[1]:=arrAxisCtrl[AxiseNo.AxisName.AnCarryingLine].Status.fSetPos;

	fActPos[2]:=arrAxisCtrl[AxiseNo.AxisName.AnCarryingUpDown].Status.fActPos;//正极送片搬运升降
	fSetPos[2]:=arrAxisCtrl[AxiseNo.AxisName.AnCarryingUpDown].Status.fSetPos;

	fActPos[3]:=arrAxisCtrl[AxiseNo.AxisName.AnCarryingWhirling].Status.fActPos;//正极送片搬运旋转
	fSetPos[3]:=arrAxisCtrl[AxiseNo.AxisName.AnCarryingWhirling].Status.fSetPos;

	fActPos[4]:=arrAxisCtrl[AxiseNo.AxisName.AnDTCarryingLine].Status.fActPos;//正极叠台搬运平移
	fSetPos[4]:=arrAxisCtrl[AxiseNo.AxisName.AnDTCarryingLine].Status.fSetPos;
	
	fActPos[5]:=arrAxisCtrl[AxiseNo.AxisName.AnDTCarryingUpDown].Status.fActPos;//正极叠台搬运升降
	fSetPos[5]:=arrAxisCtrl[AxiseNo.AxisName.AnDTCarryingUpDown].Status.fSetPos;
	
	fActPos[6]:=arrAxisCtrl[AxiseNo.AxisName.CaCarryingLine2].Status.fActPos;//负极送片搬运平移2
	fSetPos[6]:=arrAxisCtrl[AxiseNo.AxisName.CaCarryingLine2].Status.fSetPos;

	fActPos[7]:=arrAxisCtrl[AxiseNo.AxisName.CaCarryingUpDown2].Status.fActPos;//负极送片搬运升降2
	fSetPos[7]:=arrAxisCtrl[AxiseNo.AxisName.CaCarryingUpDown2].Status.fSetPos;
	
	fActPos[8]:=arrAxisCtrl[AxiseNo.AxisName.CaDTCarryingLine].Status.fActPos;//负极叠台搬运平移
	fSetPos[8]:=arrAxisCtrl[AxiseNo.AxisName.CaDTCarryingLine].Status.fSetPos;

	fActPos[9]:=arrAxisCtrl[AxiseNo.AxisName.CaDTCarryingUpDown].Status.fActPos;//负极叠台搬运升降
	fSetPos[9]:=arrAxisCtrl[AxiseNo.AxisName.CaDTCarryingUpDown].Status.fSetPos;

	fActPos[11]:=arrAxisCtrl[AxiseNo.AxisName.LeftYDUpDown].Status.fActPos;//左压刀升降
	fSetPos[11]:=arrAxisCtrl[AxiseNo.AxisName.LeftYDUpDown].Status.fSetPos;

	fActPos[12]:=arrAxisCtrl[AxiseNo.AxisName.LeftYDLine].Status.fActPos;//左压刀开合
	fSetPos[12]:=arrAxisCtrl[AxiseNo.AxisName.LeftYDLine].Status.fSetPos;
	
	fActPos[13]:=arrAxisCtrl[AxiseNo.AxisName.RightYDUpDown].Status.fActPos;//右压刀升降
	fSetPos[13]:=arrAxisCtrl[AxiseNo.AxisName.RightYDUpDown].Status.fSetPos;

	fActPos[14]:=arrAxisCtrl[AxiseNo.AxisName.RightYDLine].Status.fActPos;//右压刀开合
	fSetPos[14]:=arrAxisCtrl[AxiseNo.AxisName.RightYDLine].Status.fSetPos;	
END_IF

//判断叠台耦合中的轴是否有报警
IF 	(arrAxisCtrl[AxiseNo.AxisName.AnCarryingLine].Status.Error AND arrAxisCtrl[AxiseNo.AxisName.AnCarryingLine].Status.Coupled) OR 
		(arrAxisCtrl[AxiseNo.AxisName.AnCarryingUpDown].Status.Error AND arrAxisCtrl[AxiseNo.AxisName.AnCarryingUpDown].Status.Coupled)OR 
		(arrAxisCtrl[AxiseNo.AxisName.AnCarryingWhirling].Status.Error AND arrAxisCtrl[AxiseNo.AxisName.AnCarryingWhirling].Status.Coupled)OR
		(arrAxisCtrl[AxiseNo.AxisName.AnDTCarryingLine].Status.Error AND arrAxisCtrl[AxiseNo.AxisName.AnDTCarryingLine].Status.Coupled)OR
		(arrAxisCtrl[AxiseNo.AxisName.AnDTCarryingUpDown].Status.Error AND arrAxisCtrl[AxiseNo.AxisName.AnDTCarryingUpDown].Status.Coupled)OR
		(arrAxisCtrl[AxiseNo.AxisName.CaCarryingLine2].Status.Error AND arrAxisCtrl[AxiseNo.AxisName.CaCarryingLine2].Status.Coupled) OR 
		(arrAxisCtrl[AxiseNo.AxisName.CaCarryingUpDown2].Status.Error AND arrAxisCtrl[AxiseNo.AxisName.CaCarryingUpDown2].Status.Coupled)OR
		(arrAxisCtrl[AxiseNo.AxisName.CaDTCarryingLine].Status.Error AND arrAxisCtrl[AxiseNo.AxisName.CaDTCarryingLine].Status.Coupled)OR
		(arrAxisCtrl[AxiseNo.AxisName.CaDTCarryingUpDown].Status.Error AND arrAxisCtrl[AxiseNo.AxisName.CaDTCarryingUpDown].Status.Coupled)OR 
		(arrAxisCtrl[AxiseNo.AxisName.LeftYDLine].Status.Error AND arrAxisCtrl[AxiseNo.AxisName.LeftYDLine].Status.Coupled)OR
		(arrAxisCtrl[AxiseNo.AxisName.LeftYDUpDown].Status.Error AND arrAxisCtrl[AxiseNo.AxisName.LeftYDUpDown].Status.Coupled)OR
		(arrAxisCtrl[AxiseNo.AxisName.RightYDLine].Status.Error AND arrAxisCtrl[AxiseNo.AxisName.RightYDLine].Status.Coupled)OR
		(arrAxisCtrl[AxiseNo.AxisName.RightYDUpDown].Status.Error AND arrAxisCtrl[AxiseNo.AxisName.RightYDUpDown].Status.Coupled)OR
		(arrAxisCtrl[AxiseNo.AxisName.SEPTATCache].Status.Error AND arrAxisCtrl[AxiseNo.AxisName.SEPTATCache].Status.Coupled)OR
		(arrAxisCtrl[AxiseNo.AxisName.SEPTATLine].Status.Error AND arrAxisCtrl[AxiseNo.AxisName.SEPTATLine].Status.Coupled)OR
		(arrAxisCtrl[AxiseNo.VirAxisName.VirTailCurl].Status.Error AND arrAxisCtrl[AxiseNo.VirAxisName.VirTailCurl].Status.Coupled) THEN
		    //  (arrAxisCtrl[AxiseNo.VirAxisName.VirGM].Status.Error AND arrAxisCtrl[AxiseNo.VirAxisName.VirGM].Status.Coupled)
			arrAxisCamError:=TRUE;
ELSE
			arrAxisCamError:=FALSE;
END_IF



IF 	(NOT arrAxisCtrl[AxiseNo.AxisName.AnCarryingLine].Status.Error AND arrAxisCtrl[AxiseNo.AxisName.AnCarryingLine].Status.Enabled) AND  
	(NOT arrAxisCtrl[AxiseNo.AxisName.AnCarryingUpDown].Status.Error AND arrAxisCtrl[AxiseNo.AxisName.AnCarryingUpDown].Status.Enabled) AND  
	(NOT arrAxisCtrl[AxiseNo.AxisName.AnCarryingWhirling].Status.Error AND arrAxisCtrl[AxiseNo.AxisName.AnCarryingWhirling].Status.Enabled) AND  
	(NOT arrAxisCtrl[AxiseNo.AxisName.AnDTCarryingLine].Status.Error AND arrAxisCtrl[AxiseNo.AxisName.AnDTCarryingLine].Status.Enabled) AND  
	(NOT arrAxisCtrl[AxiseNo.AxisName.AnDTCarryingUpDown].Status.Error AND arrAxisCtrl[AxiseNo.AxisName.AnDTCarryingUpDown].Status.Enabled) AND  
	(NOT arrAxisCtrl[AxiseNo.AxisName.CaCarryingLine2].Status.Error AND arrAxisCtrl[AxiseNo.AxisName.CaCarryingLine2].Status.Enabled) AND  
	(NOT arrAxisCtrl[AxiseNo.AxisName.CaCarryingUpDown2].Status.Error AND arrAxisCtrl[AxiseNo.AxisName.CaCarryingUpDown2].Status.Enabled) AND  
	(NOT arrAxisCtrl[AxiseNo.AxisName.CaDTCarryingLine].Status.Error AND arrAxisCtrl[AxiseNo.AxisName.CaDTCarryingLine].Status.Enabled) AND  
	(NOT arrAxisCtrl[AxiseNo.AxisName.CaDTCarryingUpDown].Status.Error AND arrAxisCtrl[AxiseNo.AxisName.CaDTCarryingUpDown].Status.Enabled) AND  
	(NOT arrAxisCtrl[AxiseNo.AxisName.LeftYDLine].Status.Error AND arrAxisCtrl[AxiseNo.AxisName.LeftYDLine].Status.Enabled) AND  
	(NOT arrAxisCtrl[AxiseNo.AxisName.LeftYDUpDown].Status.Error AND arrAxisCtrl[AxiseNo.AxisName.LeftYDUpDown].Status.Enabled) AND  
	(NOT arrAxisCtrl[AxiseNo.AxisName.RightYDLine].Status.Error AND arrAxisCtrl[AxiseNo.AxisName.RightYDLine].Status.Enabled) AND  
	(NOT arrAxisCtrl[AxiseNo.AxisName.RightYDUpDown].Status.Error AND arrAxisCtrl[AxiseNo.AxisName.RightYDUpDown].Status.Enabled) AND  
	(NOT arrAxisCtrl[AxiseNo.AxisName.SEPTATCache].Status.Error AND arrAxisCtrl[AxiseNo.AxisName.SEPTATCache].Status.Enabled) AND  
	(NOT arrAxisCtrl[AxiseNo.AxisName.SEPTATLine].Status.Error AND arrAxisCtrl[AxiseNo.AxisName.SEPTATLine].Status.Enabled)   THEN
	     //(NOT arrAxisCtrl[AxiseNo.VirAxisName.VirGM].Status.Error AND arrAxisCtrl[AxiseNo.VirAxisName.VirGM].Status.Enabled)
		DTPosError[10]:=TRUE;
ELSE
		DTPosError[10]:=FALSE;
END_IF


rArrAxisCamError(CLK:=arrAxisCamError , Q=> );
IF rArrAxisCamError.Q THEN
	arrAxisCtrl[AxiseNo.VirAxisName.VirMain].Cmd.bStop:=TRUE;//主轴停止运行
	Mach_Control.DT_b.Error_tips[7]:=TRUE;//叠台有轴故障触发主虚轴停止警告
END_IF
//CCD心跳异常报警
CDD_HeartTON1(IN:=ccd.bHeartbeat  , PT:=T#2S , Q=> , ET=> );
CDD_HeartTON2(IN:= NOT  ccd.bHeartbeat  , PT:=T#2S , Q=> , ET=> );
IF (CDD_HeartTON1.Q OR CDD_HeartTON2.Q) AND NOT Mach_Control.U.CCD_ChosesHMI THEN
	Mach_Control.DT_b.Error[20]:=TRUE;//CCD通讯异常
END_IF


DT_AlarmTon[0].IN:=Mach_Control.DT_b.fWindDiameter<=Par.stDT_date.fDiameterAlarm ;
	IF  DT_AlarmTon[0].Q THEN
			//Mach_Control.DT_b.Error[24] :=TRUE;//放卷卷径报警
	END_IF

DT_AlarmTon[1].IN:=Mach_Control.An_b.An_Quantited>Mach_Control.Ca_b.Ca_Quantited ;
	IF  DT_AlarmTon[1].Q THEN
			Mach_Control.DT_b.Error[25] :=TRUE;//正极已叠片数大于负极已叠片数报警
	END_IF


DT_AlarmTon[2].IN:=NN>=2 AND NOT Mach_Control.DT_b.Error[26] ;
	IF  DT_AlarmTon[2].Q THEN
			Mach_Control.DT_b.Error[26] :=TRUE;//连续对齐度NG报警
	END_IF


IF Par.stDT_date.YD_JS_L>=Par.stDT_date.YD_SM_L THEN
	Mach_Control.DT_b.Error[28] :=TRUE;//叠台左压刀使用已经超出寿命报警
END_IF


IF Par.stDT_date.YD_JS_R>=Par.stDT_date.YD_SM_R THEN
	Mach_Control.DT_b.Error[29] :=TRUE;//叠台右压刀使用已经超出寿命报警
END_IF

IF Mach_Control.DT_b.YD_JS_L_clear THEN
	Par.stDT_date.YD_JS_L:=0;
END_IF

IF Mach_Control.DT_b.YD_JS_R_clear THEN
	Par.stDT_date.YD_JS_R:=0;
END_IF

//叠台人工确认无片，，
IF Mach_Control.DT_b.CCD_Overhang_button THEN
	Mach_Control.DT_b.OverhandResult:=3;
END_IF

(*
//检测到叠台重片，请查看是否重片
IF Mach_Control.DT_b.Error[27] AND Mach_Control.DT_b.OverhandResult=3 AND fDT_AlarmRest.Q  THEN
	Mach_Control.DT_b.Error[27]:=FALSE;
	Mach_Control.DT_b.OverhandResult:=0;
END_IF
*)




//安全门
//IF Mach_Control.U.DT_iMode=1 THEN
	Mach_Control.DT_b.Door_error[1]:=(NOT Mach_Control.se.Securitydoorswitch1 AND NOT Mach_Control.DT_b.Door_Forbidden);
	Mach_Control.DT_b.Door_error[2]:=(NOT Mach_Control.se.Securitydoorswitch2 AND NOT Mach_Control.DT_b.Door_Forbidden);
	Mach_Control.DT_b.Door_error[3]:=(NOT Mach_Control.se.Securitydoorswitch3 AND NOT Mach_Control.DT_b.Door_Forbidden);
	Mach_Control.DT_b.Door_error[4]:=(NOT Mach_Control.se.Securitydoorswitch4 AND NOT Mach_Control.DT_b.Door_Forbidden);
//END_IF

//叠片报警复位处理
rDT_AlarmRest(CLK:=Sys_Control.btn.System_Rrestbtn , Q=> );
fDT_AlarmRest(CLK:=Sys_Control.btn.System_Rrestbtn , Q=> );
IF Mach_Control.U.DT_iMode=3 THEN//在手动状态下，复位报警
		IF fDT_AlarmRest.Q AND Mach_Control.DT_b.Error[26] THEN		
					Mach_Control.DT_b.Error[26]:=FALSE;
					NN:=0;
		END_IF
		IF fDT_AlarmRest.Q AND  Mach_Control.DT_b.Error[27] AND arrAxisCtrl[AxiseNo.VirAxisName.VirMain].Status.fActPos<1  THEN
				CCD.Over.Start.iPhotoDo:=2;
				Mach_Control.DT_b.CDD_OverStart:=TRUE;
		END_IF
		IF fDT_AlarmRest.Q AND NOT Mach_Control.DT_b.Error[27] THEN
				MEMSET(ADR(Mach_Control.DT_b.Error),0,SIZEOF(Mach_Control.DT_b.Error)); // 叠台报警复位
				MEMSET(ADR(Mach_Control.DT_b.Door_error),0,SIZEOF(Mach_Control.DT_b.Door_error)); // 叠台报警复位
				arrAxisCtrl[AxiseNo.VirAxisName.VirMain].Cmd	.bStop:=FALSE;//主轴停止运行	
		END_IF
		IF fDT_AlarmRest.Q THEN
				IF 9991<=DP_Step0 AND DP_Step0<=10006 THEN
						arrAxisCtrl[AxiseNo.VirAxisName.VirMain].Cmd	.bMoveAbs:=FALSE;	
						DP_Step0:=0;
				END_IF
		END_IF				
END_IF

IF Mach_Control.DT_b.Error[12] OR Mach_Control.DT_b.Error[13] OR Mach_Control.DT_b.Error[14] OR Mach_Control.DT_b.Error[15] OR
	   Mach_Control.DT_b.Error[16] OR Mach_Control.DT_b.Error[17] OR Mach_Control.DT_b.Error[18] OR Mach_Control.DT_b.Error[19]	OR
	   Mach_Control.An_b.Error[11] OR Mach_Control.Ca_b.Error[11] THEN
	   Mach_Control.DT_b.DT_camError:=TRUE;//叠片凸轮报警，请初始化叠台后再启动
END_IF

DT_AlarmTon[3].IN:=NOT Mach_Control.se.QYcode ;
	IF  DT_AlarmTon[3].Q THEN
			Mach_Control.DT_b.Error[2] :=TRUE;//叠台储气罐真空不足报警
	END_IF

IF Mach_Control.U.DT_iMode=1 THEN
		IF NOT arrCyCtrl[arrCyNo.CylinderName.PoleInflationCy].Status.ONState OR  DT_AlarmTon[4].Q	THEN
				Mach_Control.DT_b.Error[44]:=TRUE;//自动时，张力未OK报警		
		ELSE
				;//Mach_Control.DT_b.Error[44]:=FALSE;//自动时，张力未OK报警	
		END_IF
END_IF

//计算剩余隔膜长度
rGMmanual(CLK:=Par.stDT_date.GMlength_buttonl , Q=> );
IF rGMmanual.Q THEN
   Par.stDT_date.GMlength_manual2:=Par.stDT_date.GMlength_manual2+Par.stDT_date.GMlength_manual;	
END_IF

Par.stDT_date.GMlength_act:=Par.stDT_date.GMlength_set-(DPcount*par.stDT_date.Width)/1000-(LMcount*ABS(arrAxisPar[AxiseNo.AxisName.TailCurlLine].arrTargetPoint[2]-arrAxisPar[AxiseNo.AxisName.TailCurlLine].arrTargetPoint[3]))/1000-
(NGcount*ABS(arrAxisPar[AxiseNo.AxisName.TailCurlLine].arrTargetPoint[2]-arrAxisPar[AxiseNo.AxisName.TailCurlLine].arrTargetPoint[9]))/1000-Par.stDT_date.GMlength_manual2 ;
DPGMlength:=((214*par.stDT_date.Width)+ABS(arrAxisPar[AxiseNo.AxisName.TailCurlLine].arrTargetPoint[2]-arrAxisPar[AxiseNo.AxisName.TailCurlLine].arrTargetPoint[3]))/1000;

// (*Par.stDT_date.GMlength_actMach_Control.DT_b.fWindLength_M  < DPGMlength+5 AND Mach_Control.Ca_b.Ca_Quantited <= 0*) 
//rDtUse[6](CLK:=GMlappos[4]<=Par.stDT_date.GMAngleALM);

IF  ((Mach_Control.DT_b.fWindDiameter < Par.stDT_date.fDiameterAlarm  AND NOT Mach_Control.DT_b.GMAngleALMsel ) OR
     (GMlappos[3]<=Par.stDT_date.GMAngleALM AND GMlappos[3]>0 AND Mach_Control.DT_b.fWindDiameter<100  AND  Mach_Control.DT_b.GMAngleALMsel))  AND Mach_Control.Ca_b.Ca_Quantited <= 0 AND  Mach_Control.DT_b.bTensionOK  THEN
	Mach_Control.DT_b.Error[61]:=TRUE;//剩余隔膜不能叠一个电芯，请更换隔膜	
END_IF


IF arrCyCtrl[arrCyNo.CylinderName.PoleInflationCy].Status.OFFState AND Mach_Control.DT_b.Error[61] THEN
	Par.stDT_date.GMlength_manual:=0;
	Par.stDT_date.GMlength_manual2:=0;
	DPcount:=0;
	LMcount:=0;
	NGcount:=0;
END_IF

IF DT_AlarmTon[4].Q THEN
   Mach_Control.DT_b.Error[62]:=TRUE;//自动时隔膜张力未OK
END_IF


//压刀铁氟龙计数到达设定值
IF Par.stDT_date.YD_ferrJS>=Par.stDT_date.YD_ferrset THEN
	Mach_Control.DT_b.Error[66]:=TRUE;//压刀铁氟龙计数到达设定值
END_IF
IF Mach_Control.DT_b.YD_ferrJSclear THEN
   Par.stDT_date.YD_ferrJS:=0;
 END_IF  
 
IF NOT arrAxisCtrl[AxiseNo.AxisName.DTUpDown].Status.Homed   THEN
   Mach_Control.DT_b.Error_tips[8]:=TRUE;////叠台升降未回原点提示 
ELSE
   Mach_Control.DT_b.Error_tips[8]:=FALSE;////叠台升降未回原点提示
END_IF

//压刀限位报警
IF  NOT Dietai_Gohoming  AND  (arrAxisCtrl[AxiseNo.AxisName.LeftYDUpDown].Io .biPosLimit OR arrAxisCtrl[AxiseNo.AxisName.LeftYDUpDown].Io .biNegLimit) THEN 
           Mach_Control.DT_b.Error[72]:=TRUE;//左压刀升降限位报警
END_IF		   

IF  NOT Dietai_Gohoming  AND  (arrAxisCtrl[AxiseNo.AxisName.RightYDUpDown].Io .biPosLimit OR arrAxisCtrl[AxiseNo.AxisName.RightYDUpDown].Io .biNegLimit) THEN 
           Mach_Control.DT_b.Error[73]:=TRUE;//右压刀升降限位报警
END_IF
END_ACTION

ACTION DT_Condition:

//隔膜缓存初始位置限定
arrAxisPar[AxiseNo.AxisName.SEPTATCache].arrTargetPoint[1]:=arrAxisPar[AxiseNo.AxisName.SEPTATCache].arrTargetPoint[2]+130;


Mach_Control.DT_b.iDTRunStatus;//叠台状态

IF NOT An_JumpRules[3]AND NOT An_JumpRules[4]AND NOT An_JumpRules[5]AND NOT An_JumpRules[6]AND NOT An_JumpRules[8]
	AND NOT An_JumpRules[9]AND NOT An_JumpRules[10] AND Mach_Control.U.DT_iMode=1 AND Mach_Control.An_b.JumpPiceReady THEN
	Mach_Control.DT_b.iDTRunStatus:=1;//叠台状态--自动不跳取
ELSIF An_JumpRules[1] AND Mach_Control.U.DT_iMode=1 AND Mach_Control.An_b.JumpPiceReady THEN//OR An_JumpRules[7]
	Mach_Control.DT_b.iDTRunStatus:=2;//叠台状态--自动中其他原因跳取
ELSIF An_JumpRules[2] THEN
	Mach_Control.DT_b.iDTRunStatus:=3;//叠台状态--跳取原因--手动
END_IF

(*
IF NOT Mach_Control.An_b.JumpPiceReady AND Mach_Control.U.DT_iMode=1 THEN//--------自动不跳片
	Mach_Control.DT_b.iDTRunStatus:=1;//叠台状态--自动不跳取
ELSIF Mach_Control.An_b.JumpPiceReady AND Mach_Control.U.DT_iMode=1 THEN
	Mach_Control.DT_b.iDTRunStatus:=2;//叠台状态--自动中其他原因跳取
ELSIF  Mach_Control.An_b.JumpPiceReady  AND Mach_Control.U.DT_iMode<>1 THEN//--------跳片
	Mach_Control.DT_b.iDTRunStatus:=3;//叠台状态--跳取原因--手动
END_IF
*)
//判断负极取料机械手的各轴是否在上料侧的初始位
IF 	arrAxisCtrl[AxiseNo.AxisName.CaCarryingLine2].Status.NoMoving AND arrAxisCtrl[AxiseNo.AxisName.CaCarryingLine2].Cmd.arrbRealPoint[1] AND
	arrAxisCtrl[AxiseNo.AxisName.CaCarryingUpDown2].Status.NoMoving AND arrAxisCtrl[AxiseNo.AxisName.CaCarryingUpDown2].Cmd.arrbRealPoint[4] AND
	arrAxisCtrl[AxiseNo.AxisName.CaDTCarryingLine].Status.NoMoving AND arrAxisCtrl[AxiseNo.AxisName.CaDTCarryingLine].Cmd.arrbRealPoint[1] AND
	arrAxisCtrl[AxiseNo.AxisName.CaDTCarryingUpDown].Status.NoMoving AND arrAxisCtrl[AxiseNo.AxisName.CaDTCarryingUpDown].Cmd.arrbRealPoint[4] 
	AND NOT CA_CarryingPos2 THEN	
	CA_CarryingPos1:=TRUE;//负极搬运各轴在取料方向的初始位，允许凸轮耦合
ELSE
	CA_CarryingPos1:=FALSE;
END_IF
//负极搬运各轴在放料方向的初始位，允许凸轮耦合
IF 	arrAxisCtrl[AxiseNo.AxisName.CaCarryingLine2].Status.NoMoving AND arrAxisCtrl[AxiseNo.AxisName.CaCarryingLine2].Cmd.arrbRealPoint[2] AND
	arrAxisCtrl[AxiseNo.AxisName.CaCarryingUpDown2].Status.NoMoving AND arrAxisCtrl[AxiseNo.AxisName.CaCarryingUpDown2].Cmd.arrbRealPoint[4] AND
	arrAxisCtrl[AxiseNo.AxisName.CaDTCarryingLine].Status.NoMoving AND arrAxisCtrl[AxiseNo.AxisName.CaDTCarryingLine].Cmd.arrbRealPoint[2] AND
	arrAxisCtrl[AxiseNo.AxisName.CaDTCarryingUpDown].Status.NoMoving AND arrAxisCtrl[AxiseNo.AxisName.CaDTCarryingUpDown].Cmd.arrbRealPoint[4] 
	AND NOT CA_CarryingPos1 THEN		
	CA_CarryingPos2:=TRUE;//负极搬运各轴在放料方向的初始位，允许凸轮耦合
ELSE
	CA_CarryingPos2:=FALSE;
END_IF

//判断正取料 机械手的各轴是否在上料侧的初始位
IF 	arrAxisCtrl[AxiseNo.AxisName.AnCarryingLine].Status.NoMoving AND arrAxisCtrl[AxiseNo.AxisName.AnCarryingLine].Cmd.arrbRealPoint[1] AND
	arrAxisCtrl[AxiseNo.AxisName.AnCarryingUpDown].Status.NoMoving AND arrAxisCtrl[AxiseNo.AxisName.AnCarryingUpDown].Cmd.arrbRealPoint[4] AND
	arrAxisCtrl[AxiseNo.AxisName.AnCarryingWhirling].Status.NoMoving AND arrAxisCtrl[AxiseNo.AxisName.AnCarryingWhirling].Cmd.arrbRealPoint[1] AND
	arrAxisCtrl[AxiseNo.AxisName.AnDTCarryingLine].Status.NoMoving AND arrAxisCtrl[AxiseNo.AxisName.AnDTCarryingLine].Cmd.arrbRealPoint[1] AND
	arrAxisCtrl[AxiseNo.AxisName.AnDTCarryingUpDown].Status.NoMoving AND arrAxisCtrl[AxiseNo.AxisName.AnDTCarryingUpDown].Cmd.arrbRealPoint[4] 
	AND NOT AN_CarryingPos2 THEN	
	AN_CarryingPos1:=TRUE;//正极搬运各轴在取料方向的初始位，允许凸轮耦合
ELSE
	AN_CarryingPos1:=FALSE;
END_IF
//判断正极取料 机械手的各轴是否在叠片侧的初始位
IF 	arrAxisCtrl[AxiseNo.AxisName.AnCarryingLine].Status.NoMoving AND arrAxisCtrl[AxiseNo.AxisName.AnCarryingLine].Cmd.arrbRealPoint[2] AND
	arrAxisCtrl[AxiseNo.AxisName.AnCarryingUpDown].Status.NoMoving AND arrAxisCtrl[AxiseNo.AxisName.AnCarryingUpDown].Cmd.arrbRealPoint[4] AND
	arrAxisCtrl[AxiseNo.AxisName.AnCarryingWhirling].Status.NoMoving AND arrAxisCtrl[AxiseNo.AxisName.AnCarryingWhirling].Cmd.arrbRealPoint[2] AND
	arrAxisCtrl[AxiseNo.AxisName.AnDTCarryingLine].Status.NoMoving AND arrAxisCtrl[AxiseNo.AxisName.AnDTCarryingLine].Cmd.arrbRealPoint[2] AND
	arrAxisCtrl[AxiseNo.AxisName.AnDTCarryingUpDown].Status.NoMoving AND arrAxisCtrl[AxiseNo.AxisName.AnDTCarryingUpDown].Cmd.arrbRealPoint[4] 
	AND NOT AN_CarryingPos1 THEN	
	AN_CarryingPos2:=TRUE;//正极搬运各轴在放片方向的初始位，允许凸轮耦合
ELSE
	AN_CarryingPos2:=FALSE;
END_IF

//尾卷夹隔膜平移轴在安全位，允许负极取片移动至叠片位
IF arrAxis[AxiseNo.AxisName.TailCurlSEPTALine].Status.Homed  AND arrCyCtrl[arrCyNo.CylinderName.PoleHotCutterCy].Status.OFFState AND
	 arrAxisCtrl[AxiseNo.AxisName.TailCurlSEPTALine].Status.fSetPos <= (arrAxisPar[AxiseNo.AxisName.TailCurlSEPTALine].arrTargetPoint[1]+0.5)   THEN
	TailCurlSEPTA_SafePos:=TRUE;
ELSE
	TailCurlSEPTA_SafePos:=FALSE;
END_IF



//隔膜平移定位允许
IF arrAxisCtrl[AxiseNo.AxisName.RightYDUpDown].Cmd.arrbRealPoint[1] AND arrAxisCtrl[AxiseNo.AxisName.LeftYDUpDown].Cmd.arrbRealPoint[1] THEN
arrAxisCtrl[AxiseNo.AxisName.SEPTATLine].Cmd.GoPoint_Condition[1]:=TRUE;
arrAxisCtrl[AxiseNo.AxisName.SEPTATLine].Cmd.GoPoint_Condition[2]:=TRUE;
ELSE 	
arrAxisCtrl[AxiseNo.AxisName.SEPTATLine].Cmd.GoPoint_Condition[1]:=FALSE;
arrAxisCtrl[AxiseNo.AxisName.SEPTATLine].Cmd.GoPoint_Condition[2]:=FALSE;
END_IF

//
arrAxisCtrl[AxiseNo.AxisName.SEPTATCache].Cmd.GoPoint_Condition[1]:=TRUE;


IF Mach_Control.U.DT_iMode=1 THEN
	arrDustMotor[Mach_Control.DT_b.Dust_name].bRun_FW:=TRUE;
	ELSE
	arrDustMotor[Mach_Control.DT_b.Dust_name].bRun_FW:=FALSE;		
END_IF


IF Mach_Control.U.DT_iMode=3 THEN
	Mach_Control.DT_b.Manual:=TRUE;
	ELSE
	Mach_Control.DT_b.Manual:=FALSE;	
END_IF



/////////////////////////////////////////////////////////////
/////////////////////////////////////////////////////////
////////////////////////////////////////////电机条件
//叠台升降
IF  Mach_Control.U.DT_iMode=3 OR (Mach_Control.U.WJ_iMode=1  AND TailCurlStep3=120 ) THEN
	arrAxisCtrl[AxiseNo.AxisName.DTUpDown].Cmd.Home_Condition:=TRUE;
ELSE
	arrAxisCtrl[AxiseNo.AxisName.DTUpDown].Cmd.Home_Condition:=FALSE;	
END_IF

IF  Mach_Control.U.DT_iMode=3 AND arrAxisCtrl[AxiseNo.AxisName.DTUpDown].Status.Homed AND  Mach_Control.Ca_b.Ca_Quantited =0 THEN
	arrAxisCtrl[AxiseNo.AxisName.DTUpDown].Cmd.GoPoint_Condition[1]:=TRUE;
ELSE
	arrAxisCtrl[AxiseNo.AxisName.DTUpDown].Cmd.GoPoint_Condition[1]:=FALSE;	
END_IF

IF  Mach_Control.U.DT_iMode=3 AND arrAxisCtrl[AxiseNo.AxisName.DTUpDown].Status.Homed THEN
	arrAxisCtrl[AxiseNo.AxisName.DTUpDown].Cmd.GoPoint_Condition[2]:=TRUE;
ELSE
	arrAxisCtrl[AxiseNo.AxisName.DTUpDown].Cmd.GoPoint_Condition[2]:=FALSE;	
END_IF

//叠台左压刀开合
IF  Mach_Control.U.DT_iMode=3 THEN// AND arrAxisCtrl[AxiseNo.AxisName.LeftYDUpDown].Cmd.arrbRealPoint[2]
	arrAxisCtrl[AxiseNo.AxisName.LeftYDLine].Cmd.Home_Condition:=TRUE;
ELSE
	arrAxisCtrl[AxiseNo.AxisName.LeftYDLine].Cmd.Home_Condition:=FALSE;	
END_IF

IF  Mach_Control.U.DT_iMode=3  AND //AND arrAxisCtrl[AxiseNo.AxisName.LeftYDUpDown].Cmd.arrbRealPoint[2]
	arrAxisCtrl[AxiseNo.AxisName.LeftYDLine].Status.Homed THEN
	arrAxisCtrl[AxiseNo.AxisName.LeftYDLine].Cmd.GoPoint_Condition[1]:=TRUE;
ELSE
	arrAxisCtrl[AxiseNo.AxisName.LeftYDLine].Cmd.GoPoint_Condition[1]:=FALSE;	
END_IF

IF  Mach_Control.U.DT_iMode=3 AND
	arrAxisCtrl[AxiseNo.AxisName.LeftYDLine].Status.Homed THEN//AND arrAxisCtrl[AxiseNo.AxisName.LeftYDUpDown].Cmd.arrbRealPoint[2
	arrAxisCtrl[AxiseNo.AxisName.LeftYDLine].Cmd.GoPoint_Condition[2]:=TRUE;
ELSE
	arrAxisCtrl[AxiseNo.AxisName.LeftYDLine].Cmd.GoPoint_Condition[2]:=FALSE;	
END_IF

//叠台左压刀升降
IF  Mach_Control.U.DT_iMode=3  THEN
	arrAxisCtrl[AxiseNo.AxisName.LeftYDUpDown].Cmd.Home_Condition:=TRUE;
ELSE
	arrAxisCtrl[AxiseNo.AxisName.LeftYDUpDown].Cmd.Home_Condition:=FALSE;	
END_IF

IF  Mach_Control.U.DT_iMode=3  AND arrAxisCtrl[AxiseNo.AxisName.LeftYDUpDown].Status.Homed THEN
	arrAxisCtrl[AxiseNo.AxisName.LeftYDUpDown].Cmd.GoPoint_Condition[1]:=TRUE;
ELSE
	arrAxisCtrl[AxiseNo.AxisName.LeftYDUpDown].Cmd.GoPoint_Condition[1]:=FALSE;	
END_IF

IF  Mach_Control.U.DT_iMode=3  AND arrAxisCtrl[AxiseNo.AxisName.LeftYDUpDown].Status.Homed THEN
	arrAxisCtrl[AxiseNo.AxisName.LeftYDUpDown].Cmd.GoPoint_Condition[2]:=TRUE;
ELSE
	arrAxisCtrl[AxiseNo.AxisName.LeftYDUpDown].Cmd.GoPoint_Condition[2]:=FALSE;	
END_IF

IF  Mach_Control.U.DT_iMode=3  AND arrAxisCtrl[AxiseNo.AxisName.LeftYDUpDown].Status.Homed THEN
	arrAxisCtrl[AxiseNo.AxisName.LeftYDUpDown].Cmd.GoPoint_Condition[14]:=TRUE;
ELSE
	arrAxisCtrl[AxiseNo.AxisName.LeftYDUpDown].Cmd.GoPoint_Condition[14]:=FALSE;	
END_IF

IF  Mach_Control.U.DT_iMode=3  AND arrAxisCtrl[AxiseNo.AxisName.LeftYDUpDown].Status.Homed THEN
	arrAxisCtrl[AxiseNo.AxisName.LeftYDUpDown].Cmd.GoPoint_Condition[15]:=TRUE;
ELSE
	arrAxisCtrl[AxiseNo.AxisName.LeftYDUpDown].Cmd.GoPoint_Condition[15]:=FALSE;	
END_IF
//叠台右压刀开合
IF  Mach_Control.U.DT_iMode=3  THEN//AND arrAxisCtrl[AxiseNo.AxisName.RightYDUpDown].Cmd.arrbRealPoint[2]
	arrAxisCtrl[AxiseNo.AxisName.RightYDLine].Cmd.Home_Condition:=TRUE;
ELSE
	arrAxisCtrl[AxiseNo.AxisName.RightYDLine].Cmd.Home_Condition:=FALSE;	
END_IF

IF  Mach_Control.U.DT_iMode=3  AND 
	arrAxisCtrl[AxiseNo.AxisName.RightYDLine].Status.Homed THEN//AND arrAxisCtrl[AxiseNo.AxisName.RightYDUpDown].Cmd.arrbRealPoint[2]
	arrAxisCtrl[AxiseNo.AxisName.RightYDLine].Cmd.GoPoint_Condition[1]:=TRUE;
ELSE
	arrAxisCtrl[AxiseNo.AxisName.RightYDLine].Cmd.GoPoint_Condition[1]:=FALSE;	
END_IF

IF  Mach_Control.U.DT_iMode=3 AND 
	arrAxisCtrl[AxiseNo.AxisName.RightYDLine].Status.Homed THEN//AND arrAxisCtrl[AxiseNo.AxisName.RightYDUpDown].Cmd.arrbRealPoint[2] 
	arrAxisCtrl[AxiseNo.AxisName.RightYDLine].Cmd.GoPoint_Condition[2]:=TRUE;
ELSE
	arrAxisCtrl[AxiseNo.AxisName.RightYDLine].Cmd.GoPoint_Condition[2]:=FALSE;	
END_IF

//叠台右压刀升降
IF  Mach_Control.U.DT_iMode=3  THEN
	arrAxisCtrl[AxiseNo.AxisName.RightYDUpDown].Cmd.Home_Condition:=TRUE;
ELSE
	arrAxisCtrl[AxiseNo.AxisName.RightYDUpDown].Cmd.Home_Condition:=FALSE;	
END_IF

IF  Mach_Control.U.DT_iMode=3  AND arrAxisCtrl[AxiseNo.AxisName.LeftYDUpDown].Status.Homed THEN
	arrAxisCtrl[AxiseNo.AxisName.RightYDUpDown].Cmd.GoPoint_Condition[1]:=TRUE;
ELSE
	arrAxisCtrl[AxiseNo.AxisName.RightYDUpDown].Cmd.GoPoint_Condition[1]:=FALSE;	
END_IF

IF  Mach_Control.U.DT_iMode=3  AND arrAxisCtrl[AxiseNo.AxisName.LeftYDUpDown].Status.Homed THEN
	arrAxisCtrl[AxiseNo.AxisName.RightYDUpDown].Cmd.GoPoint_Condition[2]:=TRUE;
ELSE
	arrAxisCtrl[AxiseNo.AxisName.RightYDUpDown].Cmd.GoPoint_Condition[2]:=FALSE;	
END_IF

IF  Mach_Control.U.DT_iMode=3  AND arrAxisCtrl[AxiseNo.AxisName.LeftYDUpDown].Status.Homed THEN
	arrAxisCtrl[AxiseNo.AxisName.RightYDUpDown].Cmd.GoPoint_Condition[14]:=TRUE;
ELSE
	arrAxisCtrl[AxiseNo.AxisName.RightYDUpDown].Cmd.GoPoint_Condition[14]:=FALSE;	
END_IF
IF  Mach_Control.U.DT_iMode=3  AND arrAxisCtrl[AxiseNo.AxisName.LeftYDUpDown].Status.Homed THEN
	arrAxisCtrl[AxiseNo.AxisName.RightYDUpDown].Cmd.GoPoint_Condition[15]:=TRUE;
ELSE
	arrAxisCtrl[AxiseNo.AxisName.RightYDUpDown].Cmd.GoPoint_Condition[15]:=FALSE;	
END_IF
//叠台隔膜放卷纠偏
IF  Mach_Control.U.DT_iMode=3  THEN
	arrAxisCtrl[AxiseNo.AxisName.SEPTAdeviation1].Cmd.Home_Condition:=TRUE;
ELSE
	arrAxisCtrl[AxiseNo.AxisName.SEPTAdeviation1].Cmd.Home_Condition:=FALSE;	
END_IF

IF  Mach_Control.U.DT_iMode=3  AND arrAxisCtrl[AxiseNo.AxisName.SEPTAdeviation1].Status.Homed THEN
	arrAxisCtrl[AxiseNo.AxisName.SEPTAdeviation1].Cmd.GoPoint_Condition[1]:=TRUE;
ELSE
	arrAxisCtrl[AxiseNo.AxisName.SEPTAdeviation1].Cmd.GoPoint_Condition[1]:=FALSE;	
END_IF

//叠台隔膜放卷尾部纠偏
IF  Mach_Control.U.DT_iMode=3  THEN
	arrAxisCtrl[AxiseNo.AxisName.SEPTAdeviation2].Cmd.Home_Condition:=TRUE;
ELSE
	arrAxisCtrl[AxiseNo.AxisName.SEPTAdeviation2].Cmd.Home_Condition:=FALSE;	
END_IF

IF  Mach_Control.U.DT_iMode=3  AND arrAxisCtrl[AxiseNo.AxisName.SEPTAdeviation2].Status.Homed THEN
	arrAxisCtrl[AxiseNo.AxisName.SEPTAdeviation2].Cmd.GoPoint_Condition[1]:=TRUE;
ELSE
	arrAxisCtrl[AxiseNo.AxisName.SEPTAdeviation2].Cmd.GoPoint_Condition[1]:=FALSE;	
END_IF


//叠台隔膜缓存
IF  Mach_Control.U.DT_iMode=3  THEN
	arrAxisCtrl[AxiseNo.AxisName.SEPTATCache].Cmd.Home_Condition:=TRUE;
ELSE
	arrAxisCtrl[AxiseNo.AxisName.SEPTATCache].Cmd.Home_Condition:=FALSE;	
END_IF

IF  Mach_Control.U.DT_iMode=3  AND arrAxisCtrl[AxiseNo.AxisName.SEPTATCache].Status.Homed THEN
	arrAxisCtrl[AxiseNo.AxisName.SEPTATCache].Cmd.GoPoint_Condition[1]:=TRUE;
ELSE
	arrAxisCtrl[AxiseNo.AxisName.SEPTATCache].Cmd.GoPoint_Condition[1]:=FALSE;	
END_IF

//arrAxisCtrl[AxiseNo.AxisName.SEPTATension]//张力摆杆

//叠台隔膜平移
IF  Mach_Control.U.DT_iMode=3  AND arrAxisCtrl[AxiseNo.AxisName.AnDTCarryingLine].Cmd.arrbRealPoint[1] 
    AND arrAxisCtrl[AxiseNo.AxisName.CaDTCarryingLine].Cmd.arrbRealPoint[1]
	AND arrAxisCtrl[AxiseNo.AxisName.LeftYDUpDown].Cmd.arrbRealPoint[1] 
	AND arrAxisCtrl[AxiseNo.AxisName.RightYDUpDown].Cmd.arrbRealPoint[1]    THEN
	arrAxisCtrl[AxiseNo.AxisName.SEPTATLine].Cmd.Home_Condition:=TRUE;
ELSE
	arrAxisCtrl[AxiseNo.AxisName.SEPTATLine].Cmd.Home_Condition:=FALSE;	
END_IF

IF  Mach_Control.U.DT_iMode=3 
AND arrAxisCtrl[AxiseNo.AxisName.LeftYDUpDown].Cmd.arrbRealPoint[1] 
AND arrAxisCtrl[AxiseNo.AxisName.RightYDUpDown].Cmd.arrbRealPoint[1]  AND arrAxisCtrl[AxiseNo.AxisName.AnDTCarryingLine].Cmd.arrbRealPoint[1] AND arrAxisCtrl[AxiseNo.AxisName.SEPTATLine].Status.Homed THEN
	arrAxisCtrl[AxiseNo.AxisName.SEPTATLine].Cmd.GoPoint_Condition[1]:=TRUE;
ELSE
	arrAxisCtrl[AxiseNo.AxisName.SEPTATLine].Cmd.GoPoint_Condition[1]:=FALSE;	
END_IF

IF  Mach_Control.U.DT_iMode=3 
AND arrAxisCtrl[AxiseNo.AxisName.LeftYDUpDown].Cmd.arrbRealPoint[1] 
AND arrAxisCtrl[AxiseNo.AxisName.RightYDUpDown].Cmd.arrbRealPoint[1] AND arrAxisCtrl[AxiseNo.AxisName.CaDTCarryingLine].Cmd.arrbRealPoint[1] AND arrAxisCtrl[AxiseNo.AxisName.SEPTATLine].Status.Homed  THEN
	arrAxisCtrl[AxiseNo.AxisName.SEPTATLine].Cmd.GoPoint_Condition[2]:=TRUE;
ELSE
	arrAxisCtrl[AxiseNo.AxisName.SEPTATLine].Cmd.GoPoint_Condition[2]:=FALSE;	
END_IF

//叠台隔膜放卷
IF  Mach_Control.U.DT_iMode=3 THEN
	arrAxisCtrl[AxiseNo.AxisName.SEPTAunwinding].Cmd.JogN_Condition:=TRUE;
	arrAxisCtrl[AxiseNo.AxisName.SEPTAunwinding].Cmd.JogP_Condition:=TRUE;
ELSE
	arrAxisCtrl[AxiseNo.AxisName.SEPTAunwinding].Cmd.JogN_Condition:=FALSE;	
		arrAxisCtrl[AxiseNo.AxisName.SEPTAunwinding].Cmd.JogP_Condition:=FALSE;
END_IF


Mach_Control.DTRunStatus.bJumpSync S=An_JumpRules[1] OR An_JumpRules[2] OR bDiffVel[ Par.iStationNO];//20240504 CF 前几片降速叠片不考虑同步
END_ACTION

ACTION DT_SingeMode:
		
		IF Mach_Control.DT_b.SinStepMode THEN
			DP_SinStepe:=TRUE;
		ELSE
			DP_SinStepe:=FALSE;
		END_IF
END_ACTION

ACTION GMBufferCam:

(***********************************************************************************隔膜凸轮创建V2******************************************************************************************)
(*******极片缓存电机*********)
fbCreatCamGMBuffer_L.iKeyPosTemp:=0;
fbCreatCamGMBuffer_L(
	Reset:=                              stSysState.bReset  , 
	bCreatTable:=                   fbCreatCamGMBuffer_L.bCreatTable, 
	iTable:=                            TableNo.M_GMBuffer_L , //10
	iTableGMVirDriver:=          TableNo.M_GMWind_L  , //1
	iTableGMStackCalculate:=  TableNo.M_GMLengthCalculate_L , //2
	iTableGMStackMove:=       TableNo.M_GMDanserMove_L , //3
	fMaxPos:=                           fMaxPos, 
	fMinPos:=                            fMinPos , 
    iCcwSel :=                          1 , 
	arrGMCalculateTableData:= arrDeltaGMLength_L , 

	axisSlave:=                     arrAxis[AxiseNo.VirAxisName.VirMain], 
	axisMaster:=                  arrAxis[AxiseNo.AxisName.SEPTATCache] , 
	bCreatTableDone=> , 
	bCreatTableError=> , 
	bError=>  );
fbCreatCamGMBuffer_L.bCreatTableDone;
fbCreatCamGMBuffer_L.bCreatTableError;
fbCreatCamGMBuffer_L.bError;



(*******极片缓存电机*********)
fbCreatCamGMBuffer_R.iKeyPosTemp:=0;
fbCreatCamGMBuffer_R(
	Reset:=                              stSysState.bReset  , 
	bCreatTable:=                    fbCreatCamGMBuffer_R.bCreatTable, 
	iTable:=                             TableNo.M_GMBuffer_R , //20
	iTableGMVirDriver:=           TableNo.M_GMWind_R  , //4
	iTableGMStackCalculate:=   TableNo.M_GMLengthCalculate_R , //5
	iTableGMStackMove:=         TableNo.M_GMDanserMove_R , //6
    iCcwSel :=                           2 , //2
   	fMaxPos:=                           fMaxPos, 
	fMinPos:=                            fMinPos , 
	arrGMCalculateTableData:= arrDeltaGMLength_R , 

	axisSlave:=                     arrAxis[AxiseNo.VirAxisName.VirMain], 
	axisMaster:=                  arrAxis[AxiseNo.AxisName.SEPTATCache] , 
	bCreatTableDone=> , 
	bCreatTableError=> , 
	bError=>  );
fbCreatCamGMBuffer_R.bCreatTableDone;
fbCreatCamGMBuffer_R.bCreatTableError;
fbCreatCamGMBuffer_R.bError;


(***********隔膜放卷虚轴*凸轮表**************)
fbCreatCamVirGMDriver(
	bCreatTable:=         fbCreatCamVirGMDriver.bCreatTable , 
	Reset:=                  stSysState.bReset, 
	iTable_L:=               TableNo.M_GMWind_L , //1
	iTable_R:=               TableNo.M_GMWind_R , //4

	fGMLength_L:=       arrDeltaGMLength_L[3600,1] , // (arrDeltaGMLength_L[3600,1]+arrDeltaGMLength_R[3600,1])*0.5 
	fGMLength_R:=       arrDeltaGMLength_R[3600,1] , 

